(* CODESYS project NPM_v1
   Version: 1.12

Project tree, tasks and I/O mapping:
  _750_8001_WAGO_Basic_Controller_100 : 750-8001 WAGO Basic Controller 100, WAGO, order no. 750-8001, version 1.1.0.1
    application Application
    Kbus : Kbus, WAGO, version 2.1.0.1
        unmapped channels: K-BUS diagnostics
      SC11 : 750-430, WAGO, order no. 750-430, version 2.0.0.14
          unmapped channels: _IN
      SC21 : 750-530, WAGO, order no. 750-530, version 2.0.0.15
          unmapped channels: _OUT
      SC31 : 750-459#08, WAGO, order no. 750-459, version 2.0.0.13
          unmapped channels: _IW 1, _IW 2, _IW 3, _IW 4
      SC32 : 750-459#08, WAGO, order no. 750-459, version 2.0.0.13
          unmapped channels: _IW 1, _IW 2, _IW 3, _IW 4
      SC41 : 750-658#24, WAGO, order no. 750-658, version 2.0.0.11
          unmapped channels: _INPUTCHANNEL, _OUTPUTCHANNEL
      SC42 : 750-658#24, WAGO, order no. 750-658, version 2.0.0.11
          unmapped channels: _INPUTCHANNEL, _OUTPUTCHANNEL
  _750_8212_PFC200 : 750-8212 PFC200, WAGO, order no. 750-8212, version 6.1.1.11
    application Application
      libraries: WagoAppCanLayer2, 1.6.1.4 (WAGO); BASIC, 3.3.4.0 (OSCAT); Util, 3.5.19.0 (System); CAA Memory, * (CAA Technical Workgroup)
      task FastTask (cyclic, interval 1 ms, priority 5) calls CAN_Main
      task Task (cyclic, interval 200 ms, priority 15) calls Simulate, Main
      ALGO/
        SOC/
          global variables gvSOC
          function block SOC [ST]: Calculate, CheckSOCLimits, GetSOCFromCharge, RecalibrateViaLookUpTable
          data type typSOC
        SOF/
          function block CurrentDerating [ST]: Calculate, CalculateCurves, CalculateTemperatureBasedCurrentLimit, CalculateVoltageBasedCurrentLimits, Fb_Init
          global variables gvSOF
          data type typSOF
          data type typSOF_CONFIG
          data type typSOF_CURRENT_LIMITS
          data type typSOF_CURVE
        StateEstimation/
          function block StateEstimation [ST]
      BALANCING/
        function block BAL_Dukosi [ST]: Activate, BalancingAlarm, CheckStateRequest, Deactivate, ProcessState_Balancing, ProcessState_CheckBalancing, Run, SetStateRequest, TransferStateRequest
        global variables BALANCING_CONFIG
        function block BalancingControl [ST]: Activate, CheckStateRequest, Deactivate, Process, ProcessState_Balancing, ProcessState_CheckBalancing, SetStateRequest
        data type eBAL_RETURN
        data type eBAL_STATE
        data type eBAL_STATE_REQUEST
        data type eBAL_SUB_STATE
        global variables gvBALANCING
        data type typBAL_STATE
        data type typBALANCING_CONTROL
      BMS/
        function block StringMinMax [ST]: CalculateDyeTemperatureMinMaxAverage, CalculateTemperatureMinMaxAverage, CalculateVoltageMinMaxAverage, CheckDyeTemperatureSpread, CheckTemperatureSpread, CheckVoltageSpread, Main, ValidateCellDyeTemperature, ValidateCellTemperature, ValidateCellVoltage
      function block BMS_String [ST]: GetCurrentFlowDirection, GetStringState, UpdateStringState
      BMSUtils/
        function DecodeCAN_ID [ST]
        function GetSOCFromVoltage [ST]
      CANBUS/
        function block CAN [ST]: Init, Read, UpdateCellData, Write
        global variables CAN_CONFIG
        program CAN_Main [ST]
        function block CAN_TxCurrentSensor [ST]
        function block CAN_TxDukosi [ST]
        CANUtils/
          function CAN_TO_DINT [ST]
          function CAN_TO_INT [ST]
          function CAN_TO_REAL [ST]
        data type eCAN_MESSAGE_ID
        data type eTX_STATUS
        global variables GVL_CAN_Data
        Queue/
          function block CAN_Queue [ST]: addToQueue, getFront, isEmpty, isFull, removeFromQueue
          interface ICAN_Queue: addToQueue, getFront, isEmpty, isFull, removeFromQueue
        data type typCAN_SIGNAL_RX
        data type typCAN_SIGNAL_RX_CONFIG
        data type typCAN_SIGNAL_RX_INFO
        data type typCAN_SIGNAL_TX
      CONFIG/
        global variables BAT_CELL_CONFIG
        global variables STRING_CONFIG
      data type eCANCommState
      global variables gvBMS
      global variables gvCELLS
      program Main [ST]
      function block Module [ST]
      global variables PersistentVars
      program Simulate [ST]
      data type typCAN_ID
      Types/
        CELL/
          Alarms/
            data type typCELL_ALARM_BITS
            data type uCELL_ALARMS
          Control/
            data type typBAL_CONTROL_BITS
            data type uBAL_CONTROL_BYTE
          Status/
            data type typCELL_BAL_STATUS_BITS
            data type uCELL_BAL_STATUS
          data type typCELL_ALARMS
          data type typCELL_BAL_CURRENT
          data type typCELL_BAL_STATUS
          data type typCELL_CONTROL
          data type typCELL_DYE_TEMPERATURE
          data type typCELL_MEAS
          data type typCELL_MOL_FLAG
          data type typCELL_MSL_FLAG
          data type typCELL_RSL_FLAG
          data type typCELL_TEMP
          data type typCELL_TEMPERATURE
          data type typCELL_VOLTAGE
        data type eBMS_CURRENT_FLOW_STATE
        data type eRET_VAL
        data type eSTRING_STATE
        data type NULL_REF
        data type typERROR_FLAG
        data type typMIN_MAX
        data type typSOE
        data type typSOH
        data type typSTRING_STATE
        data type typSTRING_VALUES
        data type typVoltageVsSOC
      data type typStats
      Utils/
        function BYTE_OF_DWORD [ST]
        function Compare2Arrays [ST]
        function MATH_LinearInterpolation [ST]
        function block Pulse1Sec [ST]
        function Sigmoid [ST]
        function T_PLC_MS [ST]
    Kbus : Kbus, WAGO, version 2.1.0.1
        unmapped channels: K-BUS diagnostics
      _750_658_24 : 750-658#48, WAGO, order no. 750-658, version 2.0.0.11
          unmapped channels: _INPUTCHANNEL, _OUTPUTCHANNEL
      _75x_2DI : 75x-2DI, WAGO, version 2.0.0.13
          unmapped channels: _IN
      _75x_2DO : 75x-2DO, WAGO, version 2.0.0.13
          unmapped channels: _OUT
    Serial
      COM1 : COM1, WAGO, version 0.0.0.19
  text list GlobalTextList
*)

// _750_8212_PFC200/Application/eCANCommState
{attribute 'qualified_only'}
{attribute 'strict'}
TYPE eCANCommState :
(
	INIT,
	OPEN_L2,
	CLOSE_L2,
	RESET_L2,
	CONFIG_L2,
	ALARM,
	READ,
	WRITE
);
END_TYPE

// _750_8212_PFC200/Application/typCAN_ID
TYPE typCAN_ID :
STRUCT
	P : BYTE; //Prority
	//PGN : WORD;
	ID : BYTE; //CAN type
	CA : BYTE; //Cell address
	SA : BYTE; //Station address
END_STRUCT
END_TYPE

// _750_8212_PFC200/Application/typStats
TYPE typStats :
STRUCT
	MinValue : REAL;
	MaxValue : REAL;
	AvgValue : REAL;
END_STRUCT
END_TYPE

// _750_8212_PFC200/Application/BALANCING/eBAL_RETURN
{attribute 'qualified_only'}
{attribute 'strict'}
TYPE eBAL_RETURN :
(
	BAL_OK,               
    BAL_BUSY_OK,           
    BAL_REQUEST_PENDING,   
    BAL_ILLEGAL_REQUEST,   
    BAL_INIT_ERROR, 
    BAL_OK_FROM_ERROR,
    BAL_ERROR,
    BAL_ALREADY_INITIALIZED,
    BAL_ILLEGAL_TASK_TYPE
);
END_TYPE

// _750_8212_PFC200/Application/BALANCING/eBAL_STATE
{attribute 'qualified_only'}
{attribute 'strict'}
TYPE eBAL_STATE :
(
	BAL_STATEMACH_UNINITIALIZED,
    BAL_STATEMACH_INITIALIZATION,
    BAL_STATEMACH_INITIALIZED,
    BAL_STATEMACH_CHECK_BALANCING,
    BAL_STATEMACH_BALANCE,
    BAL_STATEMACH_NO_BALANCING,
    BAL_STATEMACH_ALLOWBALANCING,
    BAL_STATEMACH_GLOBALDISABLE,
    BAL_STATEMACH_GLOBALENABLE,
    BAL_STATEMACH_UNDEFINED,
    BAL_STATEMACH_RESERVED1,
    BAL_STATEMACH_ERROR
);
END_TYPE

// _750_8212_PFC200/Application/BALANCING/eBAL_STATE_REQUEST
{attribute 'qualified_only'}
{attribute 'strict'}
TYPE eBAL_STATE_REQUEST :
(
	BAL_STATE_INIT_REQUEST,     
    BAL_STATE_ERROR_REQUEST,     
    BAL_STATE_NO_BALANCING_REQUEST, 
    BAL_STATE_ALLOWBALANCING_REQUEST, 
    BAL_STATE_GLOBAL_DISABLE_REQUEST,
    BAL_STATE_GLOBAL_ENABLE_REQUEST, 
    BAL_STATE_NO_REQUEST    
);
END_TYPE

// _750_8212_PFC200/Application/BALANCING/eBAL_SUB_STATE
{attribute 'qualified_only'}
{attribute 'strict'}
TYPE eBAL_SUB_STATE :
(
	BAL_ENTRY,       
    BAL_CHECK_IMBALANCES,
    BAL_COMPUTE_IMBALANCES,
    BAL_ACTIVATE_BALANCING,
    BAL_CHECK_LOWEST_VOLTAGE,
    BAL_CHECK_CURRENT
);
END_TYPE

// _750_8212_PFC200/Application/BALANCING/typBAL_STATE
TYPE typBAL_STATE :
STRUCT
	active : BOOL;
	balancingAllowed : BOOL;
	balancingGlobalAllowed : BOOL;
	balancingThreshold : INT;
	state : eBAL_STATE;
	substate : eBAL_SUB_STATE;
	stateRequest : eBAL_STATE_REQUEST;
END_STRUCT
END_TYPE

// _750_8212_PFC200/Application/BALANCING/typBALANCING_CONTROL
TYPE typBALANCING_CONTROL :
STRUCT
	enableBalancing : BOOL;
	threshold_mV : INT;
	request : BOOL;
	balancingState : ARRAY [1..STRING_CONFIG.BS_TOTAL_NR_OF_CELLS] OF INT;
	nrBalancedCells : INT;
END_STRUCT
END_TYPE

// _750_8212_PFC200/Application/CANBUS/eCAN_MESSAGE_ID
{attribute 'qualified_only'}
{attribute 'strict'}
TYPE eCAN_MESSAGE_ID :
(
	NONE,
	CELL_MEAS,
	CELL_TEMP,
	CELL_BAL
)BYTE;
END_TYPE

// _750_8212_PFC200/Application/CANBUS/eTX_STATUS
{attribute 'qualified_only'}
{attribute 'strict'}
TYPE eTX_STATUS :
(
	ST_CAN_TX_INIT, 
  	ST_CAN_TX_NEXT_REQ, 
  	ST_CAN_TX_BUSY, 
  	ST_CAN_TX_WRITE, 
  	ST_TCP_RECV_ERROR
);
END_TYPE

// _750_8212_PFC200/Application/CANBUS/typCAN_SIGNAL_RX
TYPE typCAN_SIGNAL_RX :
STRUCT
	Config : typCAN_SIGNAL_RX_CONFIG;
	Info : typCAN_SIGNAL_RX_INFO;
END_STRUCT
END_TYPE

// _750_8212_PFC200/Application/CANBUS/typCAN_SIGNAL_RX_CONFIG
TYPE typCAN_SIGNAL_RX_CONFIG :
STRUCT
	ID : DWORD;
	Resolution : REAL;
	Offset : REAL;
END_STRUCT
END_TYPE

// _750_8212_PFC200/Application/CANBUS/typCAN_SIGNAL_RX_INFO
TYPE typCAN_SIGNAL_RX_INFO :
STRUCT
	Data : ARRAY [1..8] OF BYTE;
	ReadRX : WagoAppCanLayer2.FbCanRx29BitFrame;
	TimeOutDelay : Standard.TON;
	pktReceived : DINT;
	pktCounter : DINT;
	pktCounter_old : DINT;
	Timpstamp : DWORD;
	previousTimestamp : DWORD;
	deltaT : DWORD;
	read : BOOL;
	newData : BOOL;
	TimeOutAlarm : BOOL;
END_STRUCT
END_TYPE

// _750_8212_PFC200/Application/CANBUS/typCAN_SIGNAL_TX
TYPE typCAN_SIGNAL_TX :
STRUCT
	CAN_NODE : __SYSTEM.IQueryInterface;
	CAN_ID : WORD;
	Data : ARRAY [1..8] OF BYTE;
END_STRUCT
END_TYPE

// _750_8212_PFC200/Application/Types/eBMS_CURRENT_FLOW_STATE
{attribute 'qualified_only'}
{attribute 'strict'}
TYPE eBMS_CURRENT_FLOW_STATE :
(
	AT_REST,
	RELAXATION,
	CHARGING,
	DISCHARGING
);
END_TYPE

// _750_8212_PFC200/Application/Types/eRET_VAL
{attribute 'qualified_only'}
{attribute 'strict'}
TYPE eRET_VAL :
(
	STD_OK,
	STD_NOT_OK
);
END_TYPE

// _750_8212_PFC200/Application/Types/eSTRING_STATE
{attribute 'qualified_only'}
{attribute 'strict'}
TYPE eSTRING_STATE :
(
	CHARGING,
	DISCHARGING,
	RELAXATION,
	AT_REST
);
END_TYPE

// _750_8212_PFC200/Application/Types/NULL_REF
TYPE NULL_REF : LINT :=0; END_TYPE

// _750_8212_PFC200/Application/Types/typERROR_FLAG
TYPE typERROR_FLAG :
STRUCT
END_STRUCT
END_TYPE

// _750_8212_PFC200/Application/Types/typMIN_MAX
TYPE typMIN_MAX :
STRUCT
	averageCellVoltage_mV : REAL;
	minimumCellVoltage_mV : REAL;
	maximumCellVoltage_mV : REAL;
	averageTemperature_degC : REAL;
	minimumTemperature_degC : REAL;
	maximumTemperature_degC : REAL;
	averageDyeTemperature_degC : REAL;
	minimumDyeTemperature_degC : REAL;
	maximumDyeTemperature_degC : REAL;
	validMeasuredCellTemperatures : INT;
	validMeasuredCellDyeTemperatures : INT;
	validMeasuredCellVoltages : INT;

END_STRUCT
END_TYPE

// _750_8212_PFC200/Application/Types/typSOE
TYPE typSOE :
STRUCT
	averageSOE_pct : REAL;
	minimumSOE_pct : REAL;
	maximumSOE_pct : REAL;
	averageSOE_Wh : REAL;
	minimumSOE_Wh : REAL;
	maximumSOE_Wh : REAL;
END_STRUCT
END_TYPE

// _750_8212_PFC200/Application/Types/typSOH
TYPE typSOH :
STRUCT
	averageSOH_pct : REAL;
	minimumSOH_pct : REAL;
	maximumSOH_pct : REAL;
END_STRUCT
END_TYPE

// _750_8212_PFC200/Application/Types/typSTRING_STATE
TYPE typSTRING_STATE :
STRUCT
	currentFlowState : eBMS_CURRENT_FLOW_STATE;
	restTime : INT;
END_STRUCT
END_TYPE

// _750_8212_PFC200/Application/Types/typSTRING_VALUES
TYPE typSTRING_VALUES :
STRUCT
	StringCurrent : REAL;
	StringVoltage : REAL;
	StringTemperature : REAL;
	StringPower : REAL;
END_STRUCT
END_TYPE

// _750_8212_PFC200/Application/Types/typVoltageVsSOC
TYPE typVoltageVsSOC :
STRUCT
	Voltage : INT;
	SOC : REAL;
END_STRUCT
END_TYPE

// _750_8212_PFC200/Application/ALGO/SOC/typSOC
TYPE typSOC :
STRUCT
	averageSOC_pct : REAL;
	minimumSOC_pct : REAL;
	maximumSOC_pct : REAL;
END_STRUCT
END_TYPE

// _750_8212_PFC200/Application/ALGO/SOF/typSOF
TYPE typSOF :
STRUCT
	recommandedContinuosChargeCurrent : REAL;
	recommandedContinuosDischargeCurrent : REAL;
	recommandedPeakChargeCurrent : REAL;
	recommandedPeakDischargeCurrent : REAL;
END_STRUCT
END_TYPE

// _750_8212_PFC200/Application/ALGO/SOF/typSOF_CONFIG
TYPE typSOF_CONFIG :
STRUCT
    maximumDischargeCurrent_mA : REAL;
    maximumChargeCurrent_mA : REAL;
    limpCurrent_mA : REAL;

    cutoffLowTemperatureDischarge_degC : REAL;
    limitLowTemperatureDischarge_degC : REAL;
    cutoffLowTemperatureCharge_degC : REAL;
    limitLowTemperatureCharge_degC : REAL;
    

    cutoffHighTemperatureDischarge_degC : REAL;
    limitHighTemperatureDischarge_degC : REAL;
    cutoffHighTemperatureCharge_degC : REAL;
    limitHighTemperatureCharge_degC : REAL;
    

    cutoffUpperCellVoltage_mV : REAL;
    limitUpperCellVoltage_mV : REAL;
    cutoffLowerCellVoltage_mV : REAL;
    limitLowerCellVoltage_mV : REAL;
END_STRUCT
END_TYPE

// _750_8212_PFC200/Application/ALGO/SOF/typSOF_CURRENT_LIMITS
TYPE typSOF_CURRENT_LIMITS :
STRUCT
	ContinuosChargeCurrent : REAL;
	ContinuosDischargeCurrent : REAL;
	PeakChargeCurrent : REAL;
	PeakDischargeCurrent : REAL;
END_STRUCT
END_TYPE

// _750_8212_PFC200/Application/ALGO/SOF/typSOF_CURVE
TYPE typSOF_CURVE :
STRUCT
	slopeLowTemperatureDischarge : REAL;   
    offsetLowTemperatureDischarge : REAL;  
    slopeHighTemperatureDischarge : REAL;  
    offsetHighTemperatureDischarge : REAL; 
    
    slopeLowTemperatureCharge : REAL;   
    offsetLowTemperatureCharge : REAL;  
    slopeHighTemperatureCharge : REAL;  
    offsetHighTemperatureCharge : REAL; 
    
    slopeUpperCellVoltage : REAL;  
    offsetUpperCellVoltage : REAL; 
    slopeLowerCellVoltage : REAL;  
    offsetLowerCellVoltage : REAL; 
END_STRUCT
END_TYPE

// _750_8212_PFC200/Application/Types/CELL/typCELL_ALARMS
TYPE typCELL_ALARMS :
STRUCT
	cellStatus : ARRAY [1..STRING_CONFIG.BS_TOTAL_NR_OF_CELLS] OF uCELL_ALARMS;
	//timeStamp : ARRAY [1..STRING_CONFIG.BS_NR_OF_MODULES, 1..STRING_CONFIG.BS_TOTAL_NR_OF_CELLS] OF DINT;
	//previousTimeStamp : ARRAY [1..STRING_CONFIG.BS_NR_OF_MODULES, 1..STRING_CONFIG.BS_TOTAL_NR_OF_CELLS] OF DINT;
END_STRUCT
END_TYPE

// _750_8212_PFC200/Application/Types/CELL/typCELL_BAL_CURRENT
TYPE typCELL_BAL_CURRENT :
STRUCT
	cellBalCurrent_mAmps : ARRAY [1..STRING_CONFIG.BS_TOTAL_NR_OF_CELLS] OF INT;
	//invalidCellBalCurrent : ARRAY [1..STRING_CONFIG.BS_NR_OF_MODULES] OF BOOL;
	nrValidCellBalCurrent : INT;
	//timeStamp : ARRAY [1..STRING_CONFIG.BS_NR_OF_MODULES, 1..STRING_CONFIG.BS_TOTAL_NR_OF_CELLS] OF DINT;
	//previousTimeStamp : ARRAY [1..STRING_CONFIG.BS_NR_OF_MODULES, 1..STRING_CONFIG.BS_TOTAL_NR_OF_CELLS] OF DINT;
END_STRUCT
END_TYPE

// _750_8212_PFC200/Application/Types/CELL/typCELL_BAL_STATUS
TYPE typCELL_BAL_STATUS :
STRUCT
	cellBalStatus : ARRAY [1..STRING_CONFIG.BS_TOTAL_NR_OF_CELLS] OF uCELL_BAL_STATUS;
	//timeStamp : ARRAY [1..STRING_CONFIG.BS_NR_OF_MODULES, 1..STRING_CONFIG.BS_TOTAL_NR_OF_CELLS] OF DINT;
	//previousTimeStamp : ARRAY [1..STRING_CONFIG.BS_NR_OF_MODULES, 1..STRING_CONFIG.BS_TOTAL_NR_OF_CELLS] OF DINT;
END_STRUCT
END_TYPE

// _750_8212_PFC200/Application/Types/CELL/typCELL_CONTROL
TYPE typCELL_CONTROL :
STRUCT
	BAL_tgtVoltage : ARRAY [1..STRING_CONFIG.BS_TOTAL_NR_OF_CELLS] OF INT;
	BAL_loadResistor : ARRAY [1..STRING_CONFIG.BS_TOTAL_NR_OF_CELLS] OF INT;
	BAL_dutyCycle : ARRAY [1..STRING_CONFIG.BS_TOTAL_NR_OF_CELLS] OF BYTE;
	BAL_watchdogUnit : ARRAY [1..STRING_CONFIG.BS_TOTAL_NR_OF_CELLS] OF BYTE;
	BAL_watchdogCounter : ARRAY [1..STRING_CONFIG.BS_TOTAL_NR_OF_CELLS] OF BYTE;
	BAL_Control : ARRAY [1..STRING_CONFIG.BS_TOTAL_NR_OF_CELLS] OF uBAL_CONTROL_BYTE;
	timeStamp : ARRAY [1..STRING_CONFIG.BS_TOTAL_NR_OF_CELLS] OF DINT;
	previousTimeStamp : ARRAY [1..STRING_CONFIG.BS_TOTAL_NR_OF_CELLS] OF DINT;
END_STRUCT
END_TYPE

// _750_8212_PFC200/Application/Types/CELL/typCELL_DYE_TEMPERATURE
TYPE typCELL_DYE_TEMPERATURE :
STRUCT
	cellDyeTemperature_deg : ARRAY [1..STRING_CONFIG.BS_TOTAL_NR_OF_CELLS] OF INT;
	invalidCellDyeTemperature : ARRAY [1..STRING_CONFIG.BS_NR_OF_MODULES] OF ULINT;
	nrValidCellDyeTemperatures :  INT;
	//timeStamp : ARRAY [1..STRING_CONFIG.BS_NR_OF_MODULES, 1..STRING_CONFIG.BS_TOTAL_NR_OF_CELLS] OF DINT;
	//previousTimeStamp : ARRAY [1..STRING_CONFIG.BS_NR_OF_MODULES, 1..STRING_CONFIG.BS_TOTAL_NR_OF_CELLS] OF DINT;
END_STRUCT
END_TYPE

// _750_8212_PFC200/Application/Types/CELL/typCELL_MEAS
TYPE typCELL_MEAS :
STRUCT
	voltage : typCELL_VOLTAGE;
	balCurrent : typCELL_BAL_CURRENT;
	cellStatus : ARRAY [1..STRING_CONFIG.BS_TOTAL_NR_OF_CELLS] OF uCELL_ALARMS;
	cellBalStatus : ARRAY [1..STRING_CONFIG.BS_TOTAL_NR_OF_CELLS] OF uCELL_BAL_STATUS;
	timeStamp : ARRAY [1..STRING_CONFIG.BS_TOTAL_NR_OF_CELLS] OF DWORD;
	previousTimeStamp : ARRAY [1..STRING_CONFIG.BS_TOTAL_NR_OF_CELLS] OF DWORD;
END_STRUCT
END_TYPE

// _750_8212_PFC200/Application/Types/CELL/typCELL_MOL_FLAG
(*Maximum operating limis*)
TYPE typCELL_MOL_FLAG :
STRUCT
	overVoltage 				: BOOL;
	underVoltage 				: BOOL;
	overTemperatureCharge 		: BOOL;
	overTemperatureDischarge 	: BOOL;
	underTemperatureCharge 		: BOOL;
	underTemperatureDischarge 	: BOOL;
	ChargeOvercurrent 			: BOOL;
	DischargeOvercurrent 		: BOOL;
END_STRUCT
END_TYPE

// _750_8212_PFC200/Application/Types/CELL/typCELL_MSL_FLAG
(*Maximum saftey limits*)
TYPE typCELL_MSL_FLAG :
STRUCT
	overVoltage 				: BOOL;
	underVoltage 				: BOOL;
	overTemperatureCharge 		: BOOL;
	overTemperatureDischarge 	: BOOL;
	underTemperatureCharge 		: BOOL;
	underTemperatureDischarge 	: BOOL;
	ChargeOvercurrent 			: BOOL;
	DischargeOvercurrent 		: BOOL;
END_STRUCT
END_TYPE

// _750_8212_PFC200/Application/Types/CELL/typCELL_RSL_FLAG
(*Recomanded saftey limits*)
TYPE typCELL_RSL_FLAG :
STRUCT
	overVoltage 				: BOOL;
	underVoltage 				: BOOL;
	overTemperatureCharge 		: BOOL;
	overTemperatureDischarge 	: BOOL;
	underTemperatureCharge 		: BOOL;
	underTemperatureDischarge 	: BOOL;
	ChargeOvercurrent 			: BOOL;
	DischargeOvercurrent 		: BOOL;
END_STRUCT
END_TYPE

// _750_8212_PFC200/Application/Types/CELL/typCELL_TEMP
TYPE typCELL_TEMP :
STRUCT
	temperature : typCELL_TEMPERATURE;
	dyeTemperature : typCELL_DYE_TEMPERATURE;
	timeStamp : ARRAY [1..STRING_CONFIG.BS_TOTAL_NR_OF_CELLS] OF DWORD;
	previousTimeStamp : ARRAY [1..STRING_CONFIG.BS_TOTAL_NR_OF_CELLS] OF DWORD;
END_STRUCT
END_TYPE

// _750_8212_PFC200/Application/Types/CELL/typCELL_TEMPERATURE
TYPE typCELL_TEMPERATURE :
STRUCT
	cellTemperature_deg : ARRAY [1..STRING_CONFIG.BS_TOTAL_NR_OF_CELLS] OF INT;
	invalidCellTemperature : ARRAY [1..STRING_CONFIG.BS_NR_OF_MODULES] OF ULINT;
	nrValidCellTemperatures :  INT;
	//timeStamp : ARRAY [1..STRING_CONFIG.BS_NR_OF_MODULES, 1..STRING_CONFIG.BS_TOTAL_NR_OF_CELLS] OF DINT;
	//previousTimeStamp : ARRAY [1..STRING_CONFIG.BS_NR_OF_MODULES, 1..STRING_CONFIG.BS_TOTAL_NR_OF_CELLS] OF DINT;
END_STRUCT
END_TYPE

// _750_8212_PFC200/Application/Types/CELL/typCELL_VOLTAGE
TYPE typCELL_VOLTAGE :
STRUCT
	stringVoltage_mV : DINT;
	//moduleVoltage_mV : ARRAY [1..STRING_CONFIG.BS_NR_OF_MODULES] OF DINT;
	cellVoltage_mV : ARRAY [1..STRING_CONFIG.BS_TOTAL_NR_OF_CELLS] OF INT;
	invalidCellVoltage : ARRAY [1..STRING_CONFIG.BS_NR_OF_MODULES] OF ULINT;
	nrValidCellVoltages : INT;
	//timeStamp : ARRAY [1..STRING_CONFIG.BS_NR_OF_MODULES, 1..STRING_CONFIG.BS_TOTAL_NR_OF_CELLS] OF DINT;
	//previousTimeStamp : ARRAY [1..STRING_CONFIG.BS_NR_OF_MODULES, 1..STRING_CONFIG.BS_TOTAL_NR_OF_CELLS] OF DINT;
END_STRUCT
END_TYPE

// _750_8212_PFC200/Application/Types/CELL/Alarms/typCELL_ALARM_BITS
TYPE typCELL_ALARM_BITS :
STRUCT
	LIM_V_MAX_OP : BIT; //Maximum operating voltage limit
	LIM_V_MIN_OP : BIT; //Minimum operating voltage limit
	LIM_V_MAX_SAFETY : BIT; //Maximum safety voltage limit
	LIM_V_MIN_SAFETY : BIT; //Minimum safety voltage limi
// 	LIM_I_DISCHARGE_DC : BIT; //Discharge current DC limit
// 	LIM_I_CHARGE_DC : BIT; //Charge current DC limit
// 	LIM_I_DISCHARGE_PULSE : BIT; //Discharge current pulse limit
// 	LIM_I_CHARGE_PULSE : BIT; //Charge current pulse limit
// 	LIM_I_DISCHARGE_PEAK : BIT; //Discharge current peak limit
// 	LIM_I_CHARGE_PEAK : BIT; //Charge current peak limit
// 	LIM_MEASUREMENT_PWM_IN_CURRENT : BIT; //Limit for measurement type PWM_IN_CURRENT
	LIM_MEASUREMENT_THERM1 : BIT; //Limit for measurement type THERM1
	HVIL_CONTACT: BIT; //HVIL_Contact
	LIM_MEASUREMENT_DTS : BIT; //Limit for measurement type DTS
	LIM_MEASUREMENT_PWM_IN_VOLTAGE : BIT; //Limit for measurement type PWM_IN_VOLTAGE
	LIM_OTHERS : BIT; //Other alarms
END_STRUCT
END_TYPE

// _750_8212_PFC200/Application/Types/CELL/Alarms/uCELL_ALARMS
TYPE uCELL_ALARMS :
UNION
	AlarmWord : WORD;
	CellAlarms : typCELL_ALARM_BITS;
END_UNION
END_TYPE

// _750_8212_PFC200/Application/Types/CELL/Control/typBAL_CONTROL_BITS
TYPE typBAL_CONTROL_BITS :
STRUCT
	BAL_enTgtVoltage : BIT; //Enable target voltage
	BAL_externalFET  : BIT; //Use external FET
END_STRUCT
END_TYPE

// _750_8212_PFC200/Application/Types/CELL/Control/uBAL_CONTROL_BYTE
TYPE uBAL_CONTROL_BYTE :
UNION
	ControlByte : BYTE;
	ControlBits : typBAL_CONTROL_BITS;
END_UNION
END_TYPE

// _750_8212_PFC200/Application/Types/CELL/Status/typCELL_BAL_STATUS_BITS
TYPE typCELL_BAL_STATUS_BITS :
STRUCT
	BAL_isActive 		: BIT; //Cell balancing in active state 
	BAL_IsStopCmd 		: BIT; //Cell balancing stopped due to balance stop command
	BAL_IsStopTgtVolt 	: BIT; //Cell balancing stopped due to target voltage reached
	BAL_isStopTgtSoc 	: BIT; //Cell balancing stopped due to target SoC reached
	BAL_isStopTgtWh 	: BIT; //Cell balancing stopped due to target watt hours reached
	BAL_isStopError 	: BIT; //Cell balancing stopped due to an error
	BAL_isStopTemp 		: BIT; //Cell balancing stopped due to an over temperature error
	BAL_isStopOther 	: BIT; //Cell balancing stopped due to any other error
END_STRUCT
END_TYPE

// _750_8212_PFC200/Application/Types/CELL/Status/uCELL_BAL_STATUS
TYPE uCELL_BAL_STATUS :
STRUCT
	StatusWord : WORD;
	BalStatus : typCELL_BAL_STATUS_BITS;
END_STRUCT
END_TYPE

// _750_8212_PFC200/Application/gvBMS
{attribute 'qualified_only'}
VAR_GLOBAL
	gvMinMax : typMIN_MAX;
	gcStringValues : typSTRING_VALUES;
	gcStringState : typSTRING_STATE;
	Fb_String : BMS_String := (StringState := gcStringState);
	StringStat : StringMinMax := (MinMaxTable := gvMinMax);
	BalancingControl : BAL_Dukosi := (DKS_BALControl := gvCells.gvCellControl, DKS_BALCurrent := gvCells.gvCellMeas.balCurrent, DKS_BALStatus := gvCells.gvCellMeas,
									  DKS_CellVoltage := gvCells.gvCellMeas.voltage, DKS_MinMax := gvMinMax, balControl := gvBalancing.gvBALANCING_CONTROL);
	
	
	Pulse1Sec : Pulse1Sec;
	
	
	
END_VAR

// _750_8212_PFC200/Application/gvCELLS
{attribute 'qualified_only'}
VAR_GLOBAL
	//Cells : typCELLS_VALUES;
	gvCellMeas : typCELL_MEAS;
	gvCellTemp : typCELL_TEMP;
	gvCellControl : typCELL_CONTROL;
// 	gvCellVoltages : typCELL_VOLTAGE;
// 	gvCellTemperatures : typCELL_TEMPERATURE;
// 	gvCellDyeTemperatures : typCELL_DYE_TEMPERATURE;
// 	gvCellAlarms : typCELL_ALARMS_1;
END_VAR

// _750_8212_PFC200/Application/PersistentVars
{attribute 'qualified_only'}
VAR_GLOBAL PERSISTENT RETAIN
	SOC : typSOC;
END_VAR

// _750_8212_PFC200/Application/BALANCING/BALANCING_CONFIG
{attribute 'qualified_only'}
VAR_GLOBAL CONSTANT
	//default value for the BAL voltage threshold 
	BAL_DEFAULT_THRESHOLD_mV : INT := 200;

	//maximum value that BAL voltage threshold may take
	BAL_MAXIMUM_THRESHOLD_mV : INT := 5000;
	
	//minimum value that BAL voltage threshold may take
	BAL_MINIMUM_THRESHOLD_mV : INT := 0; 
	
	//BAL hysteresis for voltage threshold when balancing was finished in mV
	BAL_HYSTERESIS_mV : INT := 200;
	
	//BAL lower voltage limit in MV
	BAL_LOWER_VOLTAGE_LIMIT_mV : INT := 2000;
	
	//BAL upper temperature limit
	BAL_UPPER_TEMPERATURE_LIMIT_degC : INT := 70;
	
END_VAR

// _750_8212_PFC200/Application/BALANCING/gvBALANCING
{attribute 'qualified_only'}
VAR_GLOBAL
	gvBALANCING_CONTROL : typBALANCING_CONTROL;
END_VAR

// _750_8212_PFC200/Application/CANBUS/CAN_CONFIG
{attribute 'qualified_only'}
{attribute 'global_init_slot' := '49988'}
VAR_GLOBAL
	CAN_OFFSET : DWORD := 16#80000000;
	CAN_TIMEOUT_DELAY : TIME := T#2S;
END_VAR

// _750_8212_PFC200/Application/CANBUS/GVL_CAN_Data
VAR_GLOBAL

	// typCanLayer2RxAllSchedule : typCanLayer2RxSchedule;
	arrCANDataRX: ARRAY [1..STRING_CONFIG.BS_TOTAL_NR_OF_CELLS] OF typCAN_SIGNAL_RX := [(Config := (ID := 16#98FF0101)),
																						 (Config := (ID := 16#98FF0301)),
																						 (Config := (ID := 16#98FF0501)),
																						 (Config := (ID := 16#98FF0701)),
																						 (Config := (ID := 16#98FF0901)),
																						 (Config := (ID := 16#98FF0B01)),
																						 (Config := (ID := 16#98FF0D01)),
																						 (Config := (ID := 16#98FF0F01)),
																						 (Config := (ID := 16#98FF1101)),
																						 (Config := (ID := 16#98FF1301)),
																						 (Config := (ID := 16#98FF1501)),
																						 (Config := (ID := 16#98FF1701)),
																						 (Config := (ID := 16#98FF1901)),
																						 (Config := (ID := 16#98FF1B01)),
																						 (Config := (ID := 16#98FF1D01)),
																						 (Config := (ID := 16#98FF1F01)),
																						 (Config := (ID := 16#98FF2101)),
																						 (Config := (ID := 16#98FF2301)),
																						 (Config := (ID := 16#98FF2501)),
																						 (Config := (ID := 16#98FF2701)),
																						 (Config := (ID := 16#98FF2901)),
																						 (Config := (ID := 16#98FF2B01)),
																						 (Config := (ID := 16#98FF2D01)),
																						 (Config := (ID := 16#98FF2F01)),
																						 (Config := (ID := 16#98FF3101)),
																						 (Config := (ID := 16#98FF3301)),
																						 (Config := (ID := 16#98FF3501)),
																						 (Config := (ID := 16#98FF3701)),
																						 (Config := (ID := 16#98FF3901)),
																						 (Config := (ID := 16#98FF3B01)),
																						 (Config := (ID := 16#98FF3D01)),
																						 (Config := (ID := 16#98FF3F01)),
																						 (Config := (ID := 16#98FF4101)),
																						 (Config := (ID := 16#98FF4301)),
																						 (Config := (ID := 16#98FF4501)),
																						 (Config := (ID := 16#98FF4701)),
																						 (Config := (ID := 16#98FF4901)),
																						 (Config := (ID := 16#98FF4B01)),
																						 (Config := (ID := 16#98FF4D01)),
																						 (Config := (ID := 16#98FF4F01)),
																						 (Config := (ID := 16#98FF5101)),
																						 (Config := (ID := 16#98FF5301)),
																						 (Config := (ID := 16#98FF5501)),
																						 (Config := (ID := 16#98FF5701)),
																						 (Config := (ID := 16#98FF5901)),
																						 (Config := (ID := 16#98FF5B01)),
																						 (Config := (ID := 16#98FF5D01)),
																						 (Config := (ID := 16#98FF5F01)),
																						 (Config := (ID := 16#98FF6101)),
																						 (Config := (ID := 16#98FF6301)),
																						 (Config := (ID := 16#98FF6501)),
																						 (Config := (ID := 16#98FF6701)),
																						 (Config := (ID := 16#98FF6901)),
																						 (Config := (ID := 16#98FF6B01)),
																						 (Config := (ID := 16#98FF6D01)),
																						 (Config := (ID := 16#98FF6F01)),
																						 (Config := (ID := 16#98FF7101)),
																						 (Config := (ID := 16#98FF7301)),
																						 (Config := (ID := 16#98FF7501)),
																						 (Config := (ID := 16#98FF7701)),
																						 (Config := (ID := 16#98FF7901)),
																						 (Config := (ID := 16#98FF7B01)),
																						 (Config := (ID := 16#98FF7D01)),
																						 (Config := (ID := 16#98FF7F01)),
																						 (Config := (ID := 16#98FF0301)),
																						 (Config := (ID := 16#98FF0501)),
																						 (Config := (ID := 16#98FF0701)),
																						 (Config := (ID := 16#98FF0901)),
																						 (Config := (ID := 16#98FF0B01)),
																						 (Config := (ID := 16#98FF0D01)),
																						 (Config := (ID := 16#98FF0F01)),
																						 (Config := (ID := 16#98FF1101)),
																						 (Config := (ID := 16#98FF1301)),
																						 (Config := (ID := 16#98FF1501)),
																						 (Config := (ID := 16#98FF1701)),
																						 (Config := (ID := 16#98FF1901)),
																						 (Config := (ID := 16#98FF1B01)),
																						 (Config := (ID := 16#98FF1D01)),
																						 (Config := (ID := 16#98FF1F01)),
																						 (Config := (ID := 16#98FF2101)),
																						 (Config := (ID := 16#98FF2301)),
																						 (Config := (ID := 16#98FF2501)),
																						 (Config := (ID := 16#98FF2701)),
																						 (Config := (ID := 16#98FF2901)),
																						 (Config := (ID := 16#98FF2B01)),
																						 (Config := (ID := 16#98FF2D01)),
																						 (Config := (ID := 16#98FF2F01)),
																						 (Config := (ID := 16#98FF3101)),
																						 (Config := (ID := 16#98FF3301)),
																						 (Config := (ID := 16#98FF3501)),
																						 (Config := (ID := 16#98FF3701)),
																						 (Config := (ID := 16#98FF3901)),
																						 (Config := (ID := 16#98FF3B01)),
																						 (Config := (ID := 16#98FF3D01)),
																						 (Config := (ID := 16#98FF3F01)),
																						 (Config := (ID := 16#98FF4101)),
																						 (Config := (ID := 16#98FF4301)),
																						 (Config := (ID := 16#98FF4501)),
																						 (Config := (ID := 16#98FF4701)),
																						 (Config := (ID := 16#98FF4901)),
																						 (Config := (ID := 16#98FF4B01)),
																						 (Config := (ID := 16#98FF4D01)),
																						 (Config := (ID := 16#98FF4F01)),
																						 (Config := (ID := 16#98FF5101)),
																						 (Config := (ID := 16#98FF5301)),
																						 (Config := (ID := 16#98FF5501)),
																						 (Config := (ID := 16#98FF5701)),
																						 (Config := (ID := 16#98FF5901)),
																						 (Config := (ID := 16#98FF5B01)),
																						 (Config := (ID := 16#98FF5D01)),
																						 (Config := (ID := 16#98FF5F01)),
																						 (Config := (ID := 16#98FF6101)),
																						 (Config := (ID := 16#98FF6301)),
																						 (Config := (ID := 16#98FF6501)),
																						 (Config := (ID := 16#98FF6701)),
																						 (Config := (ID := 16#98FF6901)),
																						 (Config := (ID := 16#98FF6B01)),
																						 (Config := (ID := 16#98FF6D01)),
																						 (Config := (ID := 16#98FF6F01)),
																						 (Config := (ID := 16#98FF7101)),
																						 (Config := (ID := 16#98FF7301)),
																						 (Config := (ID := 16#98FF7501)),
																						 (Config := (ID := 16#98FF7701)),
																						 (Config := (ID := 16#98FF7901)),
																						 (Config := (ID := 16#98FF7B01)),
																						 (Config := (ID := 16#98FF7D01)),
																						 (Config := (ID := 16#98FF7F01)),
																						 (Config := (ID := 16#98FF0301)),
																						 (Config := (ID := 16#98FF0501)),
																						 (Config := (ID := 16#98FF0701)),
																						 (Config := (ID := 16#98FF0901)),
																						 (Config := (ID := 16#98FF0B01)),
																						 (Config := (ID := 16#98FF0D01)),
																						 (Config := (ID := 16#98FF0F01)),
																						 (Config := (ID := 16#98FF1101)),
																						 (Config := (ID := 16#98FF1301)),
																						 (Config := (ID := 16#98FF1501)),
																						 (Config := (ID := 16#98FF1701)),
																						 (Config := (ID := 16#98FF1901)),
																						 (Config := (ID := 16#98FF1B01)),
																						 (Config := (ID := 16#98FF1D01)),
																						 (Config := (ID := 16#98FF1F01)),
																						 (Config := (ID := 16#98FF2101)),
																						 (Config := (ID := 16#98FF2301)),
																						 (Config := (ID := 16#98FF2501)),
																						 (Config := (ID := 16#98FF2701)),
																						 (Config := (ID := 16#98FF2901)),
																						 (Config := (ID := 16#98FF2B01)),
																						 (Config := (ID := 16#98FF2D01)),
																						 (Config := (ID := 16#98FF2F01)),
																						 (Config := (ID := 16#98FF3101)),
																						 (Config := (ID := 16#98FF3301)),
																						 (Config := (ID := 16#98FF3501)),
																						 (Config := (ID := 16#98FF3701)),
																						 (Config := (ID := 16#98FF3901)),
																						 (Config := (ID := 16#98FF3B01)),
																						 (Config := (ID := 16#98FF3D01)),
																						 (Config := (ID := 16#98FF3F01)),
																						 (Config := (ID := 16#98FF4101)),
																						 (Config := (ID := 16#98FF4301)),
																						 (Config := (ID := 16#98FF4501)),
																						 (Config := (ID := 16#98FF4701)),
																						 (Config := (ID := 16#98FF4901)),
																						 (Config := (ID := 16#98FF4B01)),
																						 (Config := (ID := 16#98FF4D01)),
																						 (Config := (ID := 16#98FF4F01)),
																						 (Config := (ID := 16#98FF5101)),
																						 (Config := (ID := 16#98FF5301)),
																						 (Config := (ID := 16#98FF5501)),
																						 (Config := (ID := 16#98FF5701)),
																						 (Config := (ID := 16#98FF5901)),
																						 (Config := (ID := 16#98FF5B01)),
																						 (Config := (ID := 16#98FF5D01)),
																						 (Config := (ID := 16#98FF5F01)),
																						 (Config := (ID := 16#98FF6101)),
																						 (Config := (ID := 16#98FF6301)),
																						 (Config := (ID := 16#98FF6501)),
																						 (Config := (ID := 16#98FF6701)),
																						 (Config := (ID := 16#98FF6901)),
																						 (Config := (ID := 16#98FF6B01)),
																						 (Config := (ID := 16#98FF6D01)),
																						 (Config := (ID := 16#98FF6F01)),
																						 (Config := (ID := 16#98FF7101)),
																						 (Config := (ID := 16#98FF7301)),
																						 (Config := (ID := 16#98FF7501)),
																						 (Config := (ID := 16#98FF7701)),
																						 (Config := (ID := 16#98FF7901)),
																						 (Config := (ID := 16#98FF7B01)),
																						 (Config := (ID := 16#98FF7D01)),
																						 (Config := (ID := 16#98FF7F01)),
																						 (Config := (ID := 16#98FF0301)),
																						 (Config := (ID := 16#98FF0501)),
																						 (Config := (ID := 16#98FF0701)),
																						 (Config := (ID := 16#98FF0901)),
																						 (Config := (ID := 16#98FF0B01)),
																						 (Config := (ID := 16#98FF0D01)),
																						 (Config := (ID := 16#98FF0F01)),
																						 (Config := (ID := 16#98FF1101)),
																						 (Config := (ID := 16#98FF1301)),
																						 (Config := (ID := 16#98FF1501)),
																						 (Config := (ID := 16#98FF1701)),
																						 (Config := (ID := 16#98FF1901)),
																						 (Config := (ID := 16#98FF1B01)),
																						 (Config := (ID := 16#98FF1D01))];								
	
END_VAR

// _750_8212_PFC200/Application/CONFIG/BAT_CELL_CONFIG
{attribute 'qualified_only'}
VAR_GLOBAL CONSTANT
	stateOfChargeLookupTable : ARRAY [1..10] OF typVoltageVsSOC;
	stateOfChargeLookupTableSize : UINT := SIZEOF(stateOfChargeLookupTable)/ SIZEOF(typVoltageVsSOC);
	
	CELL_TEMPERATURE_SPREAD_TOLERANCE : REAL := 10;
	CELL_VOLTAGE_SPREAD_TOLERANCE : REAL := 10;
	CELL_DYE_TEMPERATURE_SPREAD_TOLERANCE : REAL := 10;
	
	CURRENT_LEAK : REAL := 1E-6;
	CELL_NOMINAL_CAPACITY_Ah : REAL := 175; //Amps/h
	CELL_NOMINAL_ENERGY_Wh : REAL := 175; //Amps/h
	CELL_NOMINAL_CAPACITY_W : REAL := 955; //W
	CELL_NOMINAL_VOLTAGE_mV : REAL := 2300; //mW
	
	
	(*When maximum safety limit (MSL) is violated, error state is
    requested and contactors will open. When recommended safety limit
    (RSL) or maximum operating limit (MOL) is violated, the respective
    flag will be set.*)
	
	//Maximum temperature limit during discharge.
	CELL_TEMPERATURE_MAX_DISCHARGE_MSL_degC : REAL := 40;
	CELL_TEMPERATURE_MAX_DISCHARGE_RSL_degC : REAL := 39;
	CELL_TEMPERATURE_MAX_DISCHARGE_MOL_degC : REAL := 38;
	
	//Minimum temperature limit during discharge.
	CELL_TEMPERATURE_MIN_DISCHARGE_MSL_degC : REAL := -20;
	CELL_TEMPERATURE_MIN_DISCHARGE_RSL_degC : REAL := -15;
	CELL_TEMPERATURE_MIN_DISCHARGE_MOL_degC : REAL := -10;
	
	//Maximum temperature limit during charge.
	CELL_TEMPERATURE_MAX_CHARGE_MSL_degC : REAL := 40;
	CELL_TEMPERATURE_MAX_CHARGE_RSL_degC : REAL := 39;
	CELL_TEMPERATURE_MAX_CHARGE_MOL_degC : REAL := 38;
	
	//Minimum temperature limit during charge.
	CELL_TEMPERATURE_MIN_CHARGE_MSL_degC : REAL := -20;
	CELL_TEMPERATURE_MIN_CHARGE_RSL_degC : REAL := -15;
	CELL_TEMPERATURE_MIN_CHARGE_MOL_degC : REAL := -10;
	
	//Maximum voltage limit
	CELL_VOLTAGE_MAX_MSL_mV : REAL := 2750;
	CELL_VOLTAGE_MAX_RSL_mV : REAL := 2730;
	CELL_VOLTAGE_MAX_MOL_mV : REAL := 2700;
	
	//Minimum voltage limit
	CELL_VOLTAGE_MIN_MSL_mV : REAL := 2750;
	CELL_VOLTAGE_MIN_RSL_mV : REAL := 2730;
	CELL_VOLTAGE_MIN_MOL_mV : REAL := 2700;
	
	//Deep-discharge cell voltage limit.
	CELL_VOLTAGE_DEEP_DISCHARGE_mV : REAL := CELL_VOLTAGE_MIN_MSL_mV;
	
	//Maximum discharge current limit.
	CELL_CURRENT_MAX_DISCHARGE_MSL_mA : REAL := 175000;
	CELL_CURRENT_MAX_DISCHARGE_RSL_mA : REAL := 175000;
	CELL_CURRENT_MAX_DISCHARGE_MOL_mA : REAL := 175000;
	
	//Maximum charge current limit.
	CELL_CURRENT_MAX_CHARGE_MSL_mA : REAL := 175000;
	CELL_CURRENT_MAX_CHARGE_RSL_mA : REAL := 175000;
	CELL_CURRENT_MAX_CHARGE_MOL_mA : REAL := 175000;
	
END_VAR

// _750_8212_PFC200/Application/CONFIG/STRING_CONFIG
{attribute 'qualified_only'}
VAR_GLOBAL CONSTANT

	BS_NR_OF_CELLS_M1 : INT := 64;
	BS_NR_OF_CELLS_M2 : INT := 64;
	BS_NR_OF_CELLS_M3 : INT := 64;
	BS_NR_OF_CELLS_M4 : INT := 16;
	BS_NR_OF_MODULES : INT := 4;
	BS_MAX_NR_OF_CELLS_PER_MODULE : INT := 64;
	BS_NR_OF_PARALLEL_CELLS : INT := 1;
	BS_TOTAL_NR_OF_CELLS : INT := BS_NR_OF_CELLS_M1 + BS_NR_OF_CELLS_M2	+ BS_NR_OF_CELLS_M3	+ BS_NR_OF_CELLS_M4;

	BS_POSITIVE_DISCHARGE_CURRENT  : BOOL := TRUE;
	BS_REST_CURRENT_mA : INT := 200;
	BS_RELAXATION_PERIOD : INT := 5000;
	
	//Value of the balancing resistors
	BS_BALANCING_RESISTANCE_ohm : INT := 100;
	
	SOC_STRING_CAPACITY_Ah : REAL := BS_NR_OF_PARALLEL_CELLS * BAT_CELL_CONFIG.CELL_NOMINAL_CAPACITY_Ah;
	SOC_STRING_CAPACITY_mAs : REAL := SOC_STRING_CAPACITY_Ah * 3600; //mAs
	SOC_STRING_CAPACITY_As : REAL := SOC_STRING_CAPACITY_mAs/1000; //mA
	
	SOC_MAXIMUM_SOC : REAL := 100;
	SOC_MINIMUM_SOC : REAL := 0;
	
END_VAR

// _750_8212_PFC200/Application/ALGO/SOC/gvSOC
{attribute 'qualified_only'}
VAR_GLOBAL
	gvSOC : typSOC;
END_VAR

// _750_8212_PFC200/Application/ALGO/SOF/gvSOF
{attribute 'qualified_only'}
VAR_GLOBAL CONSTANT
	//Maximum current in mA in charge direction that a string can sustain.
	STRING_CURRENT_CONTINUOUS_CHARGE_mA : REAL := BAT_CELL_CONFIG.CELL_CURRENT_MAX_CHARGE_MOL_mA * STRING_CONFIG.BS_NR_OF_PARALLEL_CELLS;
	
	//Maximum current in mA in discharge direction that a string can deliver.
	STRING_CURRENT_CONTINUOUS_DISCHARGE_mA : REAL := BAT_CELL_CONFIG.CELL_CURRENT_MAX_DISCHARGE_MOL_mA * STRING_CONFIG.BS_NR_OF_PARALLEL_CELLS;
	
	//Cold temperature in °C where the derating of maximum discharge current starts
	STRING_TEMPERATURE_LOW_CUTOFF_DISCHARGE_degC : REAL := BAT_CELL_CONFIG.CELL_TEMPERATURE_MIN_DISCHARGE_MOL_degC;
	
	//Cold temperature in °C where the derating of maximum discharge current is fully applied
	STRING_TEMPERATURE_LOW_LIMIT_DISCHARGE_degC : REAL := BAT_CELL_CONFIG.CELL_TEMPERATURE_MIN_DISCHARGE_MSL_degC;
	
	//Cold temperature in °C where the derating of maximum scharge current starts
	STRING_TEMPERATURE_LOW_CUTOFF_CHARGE_degC : REAL := BAT_CELL_CONFIG.CELL_TEMPERATURE_MIN_CHARGE_MOL_degC;
	
	//Cold temperature in °C where the derating of maximum scharge current is fully applied
	STRING_TEMPERATURE_LOW_LIMIT_CHARGE_degC : REAL := BAT_CELL_CONFIG.CELL_TEMPERATURE_MIN_CHARGE_MSL_degC;
	
	//Hot temperature in °C where the derating of maximum discharge current starts
	STRING_TEMPERATURE_HIGH_CUTOFF_DISCHARGE_degC : REAL := BAT_CELL_CONFIG.CELL_TEMPERATURE_MAX_DISCHARGE_MOL_degC;
	
	//Hot temperature in °C where the derating of maximum discharge current is fully applied
	STRING_TEMPERATURE_HIGH_LIMIT_DISCHARGE_degC : REAL := BAT_CELL_CONFIG.CELL_TEMPERATURE_MAX_DISCHARGE_MSL_degC;
	
	//Hot temperature in °C where the derating of maximum dcharge current starts
	STRING_TEMPERATURE_HIGH_CUTOFF_CHARGE_degC : REAL := BAT_CELL_CONFIG.CELL_TEMPERATURE_MAX_CHARGE_MOL_degC;
	
	//Hot temperature in °C where the derating of maximum charge current is fully applied
	STRING_TEMPERATURE_HIGH_LIMIT_CHARGE_degC : REAL := BAT_CELL_CONFIG.CELL_TEMPERATURE_MAX_CHARGE_MSL_degC;
	
	//Above this voltage value string should not be exposed to full current in charge direction.
	STRING_VOLTAGE_CUTOFF_CHARGE_mV : REAL := BAT_CELL_CONFIG.CELL_VOLTAGE_MAX_MOL_mV;
	
	//Above this voltage value string should not be exposed to any current in charge direction.
	STRING_VOLTAGE_LIMIT_CHARGE_mV : REAL := BAT_CELL_CONFIG.CELL_VOLTAGE_MAX_MSL_mV;
	
	//Above this voltage value string should not be exposed to full current in discharge direction.
	STRING_VOLTAGE_CUTOFF_DISCHARGE_mV : REAL := BAT_CELL_CONFIG.CELL_VOLTAGE_MIN_MOL_mV;
	
	//Above this voltage value string should not be exposed to any current in discharge direction.
	STRING_VOLTAGE_LIMIT_DISCHARGE_mV : REAL := BAT_CELL_CONFIG.CELL_VOLTAGE_MIN_MSL_mV;
	
	//Current in mA that the string should be able to discharge when in limp mode.
	STRING_CURRENT_LIMP_mA : REAL := 20000;
		
END_VAR

VAR_GLOBAL
	
	SOF_Config: typSOF_CONFIG := (
								  maximumDischargeCurrent_mA := STRING_CURRENT_CONTINUOUS_CHARGE_mA,
								  maximumDischargeCurrent_mA := STRING_CURRENT_CONTINUOUS_DISCHARGE_mA,
								  cutoffLowTemperatureDischarge_degC := STRING_TEMPERATURE_LOW_CUTOFF_DISCHARGE_degC,
								  limitLowTemperatureDischarge_degC := STRING_TEMPERATURE_LOW_LIMIT_DISCHARGE_degC,
								  cutoffLowTemperatureCharge_degC := STRING_TEMPERATURE_LOW_CUTOFF_CHARGE_degC,
								  limitLowTemperatureCharge_degC := STRING_TEMPERATURE_LOW_LIMIT_CHARGE_degC,
								  cutoffHighTemperatureDischarge_degC := STRING_TEMPERATURE_HIGH_CUTOFF_DISCHARGE_degC,
								  limitHighTemperatureDischarge_degC := STRING_TEMPERATURE_HIGH_LIMIT_DISCHARGE_degC,
								  cutoffHighTemperatureCharge_degC := STRING_TEMPERATURE_HIGH_CUTOFF_CHARGE_degC,
								  limitHighTemperatureCharge_degC := STRING_TEMPERATURE_HIGH_LIMIT_CHARGE_degC, 
								  cutoffUpperCellVoltage_mV := STRING_VOLTAGE_CUTOFF_CHARGE_mV,
								  limitUpperCellVoltage_mV := STRING_VOLTAGE_LIMIT_CHARGE_mV,
								  cutoffLowerCellVoltage_mV := STRING_VOLTAGE_CUTOFF_DISCHARGE_mV,
								  limitLowerCellVoltage_mV := STRING_VOLTAGE_LIMIT_DISCHARGE_mV,
								  limpCurrent_mA := STRING_CURRENT_LIMP_mA);

	curveRecommandedOperatingCurrent : typSOF_CURVE;							  
								  
	SOFValues : typSOF;
	
	CurrentDerating : CurrentDerating;
END_VAR

// _750_8212_PFC200/Application/CANBUS/CAN_Main
PROGRAM CAN_Main
VAR
	BMS_CAN	: CAN;	
	CAN_TX_Queue : CAN_Queue;
	CAN_TxDukosi : CAN_TxDukosi;
END_VAR


BMS_CAN.Init(IoConfig_Globals._750_658_24);

BMS_CAN.Read(CellMeas := gvCELLS.gvCellMeas, CellTemp := gvCELLS.gvCellTemp);


CAN_TxDukosi(cellControl := gvCELLS.gvCellControl,
			 ICanQueue := CAN_TX_Queue);
			 		 
BMS_CAN.Write(ICanQueue := CAN_TX_Queue);

END_PROGRAM

// _750_8212_PFC200/Application/CANBUS/CAN_TxDukosi
FUNCTION_BLOCK CAN_TxDukosi
VAR_INPUT
	cellControl : typCELL_CONTROL;
	ICanQueue : ICAN_Queue;
END_VAR
VAR_OUTPUT
END_VAR
VAR
	c : INT;
	message : typCAN_SIGNAL_TX;
	oldData : ARRAY [1..STRING_CONFIG.BS_TOTAL_NR_OF_CELLS] OF ARRAY [1..8] OF BYTE;
END_VAR


FOR c := 1 TO STRING_CONFIG.BS_TOTAL_NR_OF_CELLS DO
	
		message.Data[1] := MEM.HighByte(wValue := TO_WORD(cellControl.BAL_tgtVoltage[c]));
		message.Data[2] := MEM.LowByte(wValue := TO_WORD(cellControl.BAL_tgtVoltage[c]));
		message.Data[3] := MEM.HighByte(wValue := TO_WORD(cellControl.BAL_loadResistor[c]));
		message.Data[4] := MEM.LowByte(wValue := TO_WORD(cellControl.BAL_loadResistor[c]));
		message.Data[5] := cellControl.BAL_dutyCycle[c];
		message.Data[6] := cellControl.BAL_watchdogUnit[c];
		message.Data[7] := cellControl.BAL_watchdogCounter[c];
		message.Data[8] := cellControl.BAL_Control[c].ControlByte;
		
		IF NOT ICanQueue.isFull() THEN
			IF Compare2Arrays(message.Data, oldData[c]) THEN
				message.CAN_ID := TO_WORD(4000 + c);
				ICanQueue.addToQueue(message);
				oldData[c] := message.Data;
			END_IF
		END_IF

END_FOR

END_FUNCTION_BLOCK

// _750_8212_PFC200/Application/Utils/Compare2Arrays
FUNCTION Compare2Arrays : BOOL
VAR_INPUT
	x : ARRAY [*] OF BYTE;
	y : ARRAY [*] OF BYTE;
END_VAR
VAR
	size_x : DINT;
	start_x : DINT;
	size_y : DINT;
	start_y	 : DINT;
	diff : BYTE;
	idx : DINT;
END_VAR


size_x := UPPER_BOUND(x,1);
start_x := LOWER_BOUND(x,1);
size_y := UPPER_BOUND(y,1);
start_y := LOWER_BOUND(y,1);

Compare2Arrays := FALSE;
diff := 0;

IF size_x <> size_y THEN
	RETURN;
END_IF

FOR idx := start_x TO size_x DO
	
	diff := diff OR (x[idx] - y[idx]);

END_FOR

IF (diff <> 0) THEN
	Compare2Arrays := TRUE;
END_IF

END_FUNCTION

// _750_8212_PFC200/Application/CANBUS/Queue/ICAN_Queue
INTERFACE ICAN_Queue

METHOD addToQueue : eRET_VAL
VAR_INPUT
	item : typCAN_SIGNAL_TX;
END_VAR
END_METHOD

METHOD getFront : typCAN_SIGNAL_TX
VAR_INPUT
END_VAR
END_METHOD

METHOD isEmpty : BOOL
VAR_INPUT
END_VAR
END_METHOD

METHOD isFull : BOOL
VAR_INPUT
END_VAR
END_METHOD

METHOD removeFromQueue : eRET_VAL
VAR_INPUT
END_VAR
VAR
END_VAR
END_METHOD

END_INTERFACE

// _750_8212_PFC200/Application/CANBUS/CAN
//{attribute 'global_init_slot' := '50000'}
FUNCTION_BLOCK CAN
VAR_INPUT
END_VAR
VAR_IN_OUT
	
END_VAR
VAR_OUTPUT
END_VAR
VAR
	
	m_CAN_OpenL2 : WagoAppCanLayer2.FbCanL2Open := (udiBaudrate := 500000);
	m_CAN_CloseL2 : WagoAppCanLayer2.FbCanL2Close;
	m_CAN_ResetL2 : WagoAppCanLayer2.FbCanL2Reset;
	m_CAN_Config : WagoSysModule_75x_658.FbModuleConfigurationAndStatus;
	m_CommState : INT;
	m_Bitrate : INT;
	m_Mode : INT;
	m_29BitEnabled : BOOL;
	m_SdoEnabled : BOOL;
	m_DiagOverMbx0Enabled : BOOL;
	m_ConfigData : WagoSysModule_75x_658.WagoTypesModule_75x_658.typFullConfiguration;
	m_DiagnosisReset: BOOL;
	m_CommunicationReset : BOOL;
	I_WagoSysTypeBase : WagoAppCanLayer2.WagoTypesCan.I_WagoSysCanBase;
	I_ModuleExtended : WagoSysModule_75x_658.I_WagoModule_75x_658Extended;
	m_Init : BOOL;
	m_CAN_ReadWriteEnabled : BOOL;
	m_RX : WagoAppCanLayer2.FbCanRx29BitFrameAll;
	m_TX : WagoAppCanLayer2.FbCanTx29BitFrame;
	m_Read : BOOL;
	m_Write : BOOL;
	m_TXState : INT;
	
	//c : INT;
END_VAR
VAR_TEMP
	
END_VAR

METHOD Init
VAR_INPUT
	Port : __SYSTEM.IQueryInterface;
END_VAR
IF NOT m_Init THEN
	//Port := IoConfig_Globals._750_658_24;
	__QUERYINTERFACE(Port, I_WagoSysTypeBase);
	__QUERYINTERFACE(Port, I_ModuleExtended);
	m_Init := TRUE;
END_IF;
	
CASE m_CommState OF 
	
eCANCommState.INIT:
	m_CommState := eCANCommState.OPEN_L2;
	
eCANCommState.OPEN_L2:
	IF NOT m_CAN_OpenL2.xValid AND NOT m_CAN_OpenL2.xBusy THEN
		m_CAN_OpenL2.xEnable := TRUE;
	ELSIF m_CAN_OpenL2.xValid AND NOT m_CAN_OpenL2.xError THEN
		m_CAN_ReadWriteEnabled := TRUE;
	ELSIF m_CAN_OpenL2.xError THEN
		m_CAN_ReadWriteEnabled := FALSE;
		m_CAN_OpenL2.xEnable := FALSE;	
		m_CommState := eCANCommState.CLOSE_L2;
	END_IF;	

eCANCommState.CLOSE_L2:
	m_CAN_CloseL2.xExecute := TRUE;
	IF m_CAN_CloseL2.xDone THEN
		m_CommState := eCANCommState.RESET_L2;
		m_CAN_CloseL2.xExecute := FALSE;
	END_IF
	
eCANCommState.RESET_L2:	
	m_CAN_ResetL2.xExecute := TRUE;
	IF m_CAN_ResetL2.xDone THEN
		m_CommState := eCANCommState.OPEN_L2;
		m_CAN_ResetL2.xExecute := FALSE;
	END_IF

eCANCommState.CONFIG_L2:
	m_Bitrate := 5;
	m_Mode := 1;
	m_29BitEnabled := TRUE;
	m_SdoEnabled := FALSE;
	m_DiagOverMbx0Enabled := TRUE;

	IF NOT m_CAN_Config.xBusy AND NOT m_CAN_Config.xDone THEN
		m_CAN_Config.xExecute := TRUE;
		m_CAN_Config.xWriteRead := TRUE;
		m_CAN_Config.xSaveValues := TRUE;
	ELSIF NOT m_CAN_Config.xBusy AND m_CAN_Config.xDone	THEN
		m_CAN_Config.xExecute := FALSE;
		m_CAN_Config.xWriteRead := FALSE;
		m_CAN_Config.xSaveValues := FALSE;
		m_CommState := eCANCommState.READ;
	END_IF
	
END_CASE

m_CAN_OpenL2(I_Port := I_WagoSysTypeBase,
			 udiBaudrate := 500000);

m_CAN_CloseL2(
	I_Port:= I_WagoSysTypeBase);			 

m_CAN_ResetL2(
	I_Port:= I_WagoSysTypeBase);
			 
m_CAN_Config(
	I_Port:= I_ModuleExtended, 
	eBitrate:= m_Bitrate, 
	eMode:= m_Mode, 
	x29BitEnabled:= m_29BitEnabled, 
	xSdoEnabled:= m_SdoEnabled, 
	xDiagOverMbx0Enabled:= m_DiagOverMbx0Enabled, 
	typConfigData:= m_ConfigData, 
	xDiagnosisReset:= m_DiagnosisReset, 
	xCommunicationReset:= m_CommunicationReset);
END_METHOD

METHOD Read
VAR_INPUT 
	CellMeas : REFERENCE TO typCELL_MEAS;
	CellTemp : REFERENCE TO typCELL_TEMP;
END_VAR

VAR
	_idx : INT;
END_VAR

GVL_CAN_Data.arrCANDataRX[1].Info.TimeOutDelay(	IN := TRUE,
					   							PT := CAN_CONFIG.CAN_TIMEOUT_DELAY,
					   							Q => GVL_CAN_Data.arrCANDataRX[1].Info.TimeOutAlarm);	 

m_RX(xEnable := m_CAN_ReadWriteEnabled,
	 I_Port := I_WagoSysTypeBase,
	 xRxTrigger := m_Read);

IF NOT m_Read THEN
	m_Read := TRUE;
END_IF
							 
// GVL_CAN_Data.arrCANDataRX[1].Info.Timpstamp := T_PLC_MS();										 
// //IF m_pktCounter <> m_oldPktCounter THEN
// 	IF GVL_CAN_Data.arrCANDataRX[1].Config.ID = m_RX.dwRxId + CAN_CONFIG.CAN_OFFSET THEN
// 			GVL_CAN_Data.arrCANDataRX[1].Info.TimeOutDelay(IN := FALSE);
// 			GVL_CAN_Data.arrCANDataRX[1].Info.Data := m_RX.aRxBuffer;
// 			GVL_CAN_Data.arrCANDataRX[1].Info.pktReceived := m_RX.bRxNBytes;// + Data.Info.pktReceived;	
// 			GVL_CAN_Data.arrCANDataRX[1].Info.deltaT := GVL_CAN_Data.arrCANDataRX[1].Info.Timpstamp - GVL_CAN_Data.arrCANDataRX[1].Info.previousTimestamp;
// 			GVL_CAN_Data.arrCANDataRX[1].Info.previousTimestamp := GVL_CAN_Data.arrCANDataRX[1].Info.Timpstamp;
// 			GVL_CAN_Data.arrCANDataRX[1].Info.pktCounter_old := GVL_CAN_Data.arrCANDataRX[1].Info.pktReceived;
// 	END_IF
	
UpdateCellData(m_RX.dwRxId, m_Rx.aRxBuffer, CellMeas, CellTemp);	


//END_IF
END_METHOD

METHOD PRIVATE UpdateCellData
VAR_INPUT
	CanID : DWORD;
	CanMessage : ARRAY [1..8] OF BYTE;
	CellMeas : REFERENCE TO typCELL_MEAS;
	CellTemp : REFERENCE TO typCELL_TEMP;
END_VAR
VAR
	_DecodedCAN : typCAN_ID;
	_CellIdx : INT;
END_VAR

_DecodedCAN := DecodeCAN_ID(CanID);
_CellIdx := TO_INT(STRING_CONFIG.BS_MAX_NR_OF_CELLS_PER_MODULE * (_DecodedCAN.SA - 1) + _DecodedCAN.CA);


CASE _DecodedCAN.ID OF
	
	eCAN_MESSAGE_ID.CELL_MEAS:
		CellMeas.voltage.cellVoltage_mV[_CellIdx] := CAN_TO_INT(StartByte := 1, Data := ADR(CanMessage));
		CellMeas.balCurrent.cellBalCurrent_mAmps[_CellIdx] := CAN_TO_INT(StartByte := 3, Data := ADR(CanMessage));
		CellMeas.cellStatus[_CellIdx].AlarmWord := TO_WORD(CAN_TO_INT(StartByte := 5, Data := ADR(CanMessage)));
		CellMeas.cellBalStatus[_CellIdx].StatusWord := TO_WORD(CAN_TO_INT(StartByte := 7, Data := ADR(CanMessage)));
		CellMeas.timeStamp[_CellIdx] := T_PLC_MS();
		CellMeas.previousTimeStamp[_CellIdx] := CellMeas.timeStamp[_CellIdx];
	
	eCAN_MESSAGE_ID.CELL_TEMP:
		CellTemp.temperature.cellTemperature_deg[_CellIdx] := CAN_TO_INT(StartByte := 1, Data := ADR(CanMessage));	
		CellTemp.DyeTemperature.cellDyeTemperature_deg[_CellIdx] := CAN_TO_INT(StartByte := 3, Data := ADR(CanMessage));	
		CellTemp.timeStamp[_CellIdx] := T_PLC_MS();
		CellTemp.previousTimeStamp[_CellIdx] := CellTemp.timeStamp[_CellIdx];
END_CASE
END_METHOD

METHOD Write
VAR_INPUT
	ICanQueue : ICAN_Queue;
END_VAR
VAR
	canRxSignal : typCAN_SIGNAL_TX;
END_VAR

IF ICanQueue.isEmpty() THEN
	RETURN;
END_IF 

CASE m_TXState OF
	
	eTX_STATUS.ST_CAN_TX_INIT:
		IF m_CAN_ReadWriteEnabled THEN
			m_TXState := eTX_STATUS.ST_CAN_TX_NEXT_REQ;
		END_IF

	eTX_STATUS.ST_CAN_TX_NEXT_REQ:

		canRxSignal := ICanQueue.getFront();
		m_TXState := eTX_STATUS.ST_CAN_TX_WRITE;
		m_Write := TRUE;
		
	eTX_STATUS.ST_CAN_TX_WRITE:
		IF NOT m_Write AND NOT m_TX.xError AND m_TX.xValid THEN
			m_TXState := eTX_STATUS.ST_CAN_TX_NEXT_REQ;	
			ICanQueue.removeFromQueue();
		END_IF
		
END_CASE



m_TX(xEnable := m_CAN_ReadWriteEnabled,
	 xTxTrigger := m_Write,
	 I_Port := I_WagoSysTypeBase,
	 dwCanId := canRxSignal.CAN_ID,
	 aTxBuffer := canRxSignal.Data,
	 bTxNBytes := 8);
END_METHOD

END_FUNCTION_BLOCK

// _750_8212_PFC200/Application/Utils/T_PLC_MS
FUNCTION T_PLC_MS : DWORD
VAR CONSTANT
	debug : BOOL := 0;
	N : INT := 0;
	offset : DWORD := 0;
END_VAR
VAR
	tx : TIME;
END_VAR

(*
version 1.2	16. nov 2008
programmer 	hugo
tested by	oscat

T_PLC_MS reads the internal PLC timer and return the time, it has the advantage to be able to set a debug mode 
and speed up the counter to test the plc timer overrun which occurs every 50 days respectively 25 days at siemens S7
this routine also allows to correct the behavior of s7 where the internal plc counter will not count all 32 bits.

*)

tx := TIME();
T_PLC_MS := TIME_TO_DWORD(Tx);

IF debug THEN
	T_PLC_MS := (SHL(T_PLC_MS,N) OR SHL(DWORD#1,N)-1) + OFFSET;
END_IF;

END_FUNCTION

// _750_8212_PFC200/Application/BMSUtils/DecodeCAN_ID
FUNCTION DecodeCAN_ID : typCAN_ID
VAR_INPUT
	CAN_ID : DWORD;
END_VAR
VAR
	_dwPGN : DWORD;
END_VAR

// 
// DecodeCAN_ID.SA := DWORD_TO_BYTE(SHR(CAN_ID,SHL(0,3)));
// _dwPGN := SHL(CAN_ID, 8);
// _dwPGN := SHR(_dwPGN, 8);
// _dwPGN := SHR(_dwPGN, 8);
// DecodeCAN_ID.PGN := TO_WORD(_dwPGN);
// DecodeCAN_ID.P := DWORD_TO_BYTE(SHR(CAN_ID,SHL(3,3)));

DecodeCAN_ID.SA := BYTE_OF_DWORD(CAN_ID, 0);
DecodeCAN_ID.CA := BYTE_OF_DWORD(CAN_ID, 1);
DecodeCAN_ID.ID := BYTE_OF_DWORD(CAN_ID, 2);
DecodeCAN_ID.P := BYTE_OF_DWORD(CAN_ID, 3);

END_FUNCTION

// _750_8212_PFC200/Application/Utils/BYTE_OF_DWORD
FUNCTION BYTE_OF_DWORD : BYTE
VAR_INPUT
	in : DWORD;
	N : BYTE;
END_VAR


(*
version 1.2	30. oct. 2008
programmer 	hugo
tested by	oscat

this function extracts a single byte from the nth position from right (right is lowest byte) 
the lower byte (starting with Bit0 from in) is selected with N=0.
*)

BYTE_OF_DWORD := DWORD_TO_BYTE(SHR(in,SHL(n,3)));

(* revision history
hm	17. jan 2007	rev 1.0
	original version

hm	2. jan 2008		rev 1.1
	improved performance

hm	30. oct. 2008	rev 1.2
	improved performance
*)

END_FUNCTION

// _750_8212_PFC200/Application/CANBUS/CANUtils/CAN_TO_INT
FUNCTION CAN_TO_INT : INT
VAR_INPUT
	StartByte : INT;
	Data : POINTER TO ARRAY[1..8] OF BYTE;
END_VAR
VAR
	b0 : BYTE;
    b1 : BYTE;
END_VAR

IF (Data = 0) THEN RETURN; END_IF;

b0 := Data^[StartByte];
b1 := Data^[StartByte+1];

CAN_TO_INT := TO_INT(SHL(BYTE_TO_WORD(b1),8) OR BYTE_TO_WORD(B0));

END_FUNCTION

// _750_8212_PFC200/Application/CANBUS/Queue/CAN_Queue
FUNCTION_BLOCK CAN_Queue IMPLEMENTS ICAN_Queue
VAR_INPUT
END_VAR
VAR_OUTPUT
END_VAR
VAR
	buffer : ARRAY[0..MAX_ELEMENTS-1] OF typCAN_SIGNAL_TX;
	front : INT := -1;
	rear : INT := -1;
	size : INT := MAX_ELEMENTS;
	stop: INT;
	test: INT;
END_VAR
VAR CONSTANT
	MAX_ELEMENTS : INT := 50;
END_VAR

METHOD addToQueue : eRET_VAL
VAR_INPUT
	item : typCAN_SIGNAL_TX;
END_VAR

VAR
	
END_VAR
addToQueue := eRET_VAL.STD_NOT_OK;
IF (isFull()) THEN
	RETURN;
ELSIF (front = -1) THEN
	front := rear := 0;
	buffer[rear] := item;
ELSIF (rear = size - 1 AND front <> 0) THEN
	rear := 0;
	buffer[rear] := item;
ELSE
	rear := rear + 1;
	buffer[rear] := item;
END_IF

addToQueue := eRET_VAL.STD_OK;
END_METHOD

METHOD getFront : typCAN_SIGNAL_TX
VAR_INPUT
END_VAR
IF isEmpty() THEN
	RETURN;
END_IF
IF (front = -1) THEN
	front := 0;
END_IF

getFront := buffer[front];
END_METHOD

METHOD isEmpty : BOOL
VAR_INPUT
END_VAR
isEmpty := (front = -1);
END_METHOD

METHOD isFull : BOOL
VAR_INPUT
END_VAR
isFull := (((front = 0) AND (rear = size - 1)) OR ((rear + 1) MOD size = front));
END_METHOD

METHOD removeFromQueue : eRET_VAL
VAR_INPUT
END_VAR
VAR
	elem : typCAN_SIGNAL_TX;
END_VAR
removeFromQueue := eRET_VAL.STD_NOT_OK;
IF (isEmpty()) THEN
	RETURN;
END_IF

elem := buffer[front];
IF (front = rear) THEN
	front := -1;
	rear := -1;
ELSIF (front = size - 1) THEN
	front := 0;
ELSE 
	front := front + 1;
END_IF

removeFromQueue := eRET_VAL.STD_OK;
END_METHOD

END_FUNCTION_BLOCK

// _750_8212_PFC200/Application/Simulate
PROGRAM Simulate
VAR
	c : INT;
	simVoltage : BOOL;
END_VAR

IF simVoltage THEN
	
	FOR c := 1 TO STRING_CONFIG.BS_TOTAL_NR_OF_CELLS DO
		gvCELLS.gvCellMeas.voltage.cellVoltage_mV[c] := 2000;
	END_FOR
	simVoltage := FALSE;
END_IF

END_PROGRAM

// _750_8212_PFC200/Application/Main
PROGRAM Main
VAR
xInit : BOOL;

END_VAR


IF xInit THEN
	gvBMS.BalancingControl.SetStateRequest(stateRequest := eBAL_STATE_REQUEST.BAL_STATE_ALLOWBALANCING_REQUEST);
	gvBMS.BalancingControl.SetStateRequest(stateRequest := eBAL_STATE_REQUEST.BAL_STATE_GLOBAL_ENABLE_REQUEST);
ELSE
	gvBMS.BalancingControl.SetStateRequest(stateRequest := eBAL_STATE_REQUEST.BAL_STATE_GLOBAL_DISABLE_REQUEST);
	gvBMS.BalancingControl.SetStateRequest(stateRequest := eBAL_STATE_REQUEST.BAL_STATE_GLOBAL_DISABLE_REQUEST);
END_IF

gvBMS.StringStat.Main();
gvSOF.CurrentDerating.Calculate();
gvBMS.BalancingControl.Run();
gvBMS.Pulse1Sec();

END_PROGRAM

// _750_8212_PFC200/Application/BALANCING/BalancingControl
FUNCTION_BLOCK BalancingControl
VAR_INPUT
	cellVoltage : REFERENCE TO typCELL_VOLTAGE;
	minMax : REFERENCE TO typMIN_MAX;
	balControl : REFERENCE TO typBALANCING_CONTROL;
END_VAR
VAR_OUTPUT
END_VAR
VAR
	bal_State : typBAL_STATE;
END_VAR

METHOD Activate : BOOL
VAR_INPUT

END_VAR
VAR
	cellBalancingCurrent : REAL;
	difference : INT;
	nrBalancedCells : INT;
	c : INT;
	finished : BOOL;
	minVoltage : REAL;
END_VAR

finished := TRUE;
minVoltage := minMax.minimumCellVoltage_mV;

FOR c := 1 TO STRING_CONFIG.BS_TOTAL_NR_OF_CELLS DO
	IF cellVoltage.cellVoltage_mV[c] > (minVoltage + bal_State.balancingThreshold) THEN
		balControl.balancingState[c] := 1;
		finished := FALSE;
		bal_State.balancingThreshold := balControl.threshold_mV;
		bal_state.active := TRUE;
		balControl.enableBalancing := TRUE;
		nrBalancedCells := nrBalancedCells + 1;
	ELSE
		balControl.balancingState[c] := 0;
	END_IF
END_FOR

balControl.nrBalancedCells := nrBalancedCells;

Activate := finished;
END_METHOD

METHOD CheckStateRequest : eBAL_RETURN
VAR_INPUT
	CurrentState : REFERENCE TO typBAL_STATE;
	stateRequest : eBAL_STATE_REQUEST;
END_VAR
IF (stateRequest = eBAL_STATE_REQUEST.BAL_STATE_ERROR_REQUEST) THEN
	CheckStateRequest := eBAL_RETURN.BAL_OK;
	RETURN;
END_IF

IF (stateRequest = eBAL_STATE_REQUEST.BAL_STATE_GLOBAL_ENABLE_REQUEST) THEN
	CurrentState.balancingGlobalAllowed := TRUE;
	CheckStateRequest := eBAL_RETURN.BAL_OK;
	RETURN;
END_IF

IF (stateRequest = eBAL_STATE_REQUEST.BAL_STATE_GLOBAL_DISABLE_REQUEST) THEN
	CurrentState.balancingGlobalAllowed := FALSE;
	CheckStateRequest := eBAL_RETURN.BAL_OK;
	RETURN;
END_IF

IF (stateRequest = eBAL_STATE_REQUEST.BAL_STATE_NO_BALANCING_REQUEST) OR (stateRequest = eBAL_STATE_REQUEST.BAL_STATE_ALLOWBALANCING_REQUEST) THEN
	CheckStateRequest := eBAL_RETURN.BAL_OK;
	RETURN;
END_IF

IF (CurrentState.stateRequest = eBAL_STATE_REQUEST.BAL_STATE_NO_REQUEST) THEN
	IF (stateRequest = eBAL_STATE_REQUEST.BAL_STATE_INIT_REQUEST) THEN
		IF (CurrentState.state = eBAL_STATE.BAL_STATEMACH_UNINITIALIZED) THEN
			CheckStateRequest := eBAL_RETURN.BAL_OK;
			RETURN;
		ELSE
			CheckStateRequest := eBAL_RETURN.BAL_ALREADY_INITIALIZED;
			RETURN;
		END_IF
	ELSE
		CheckStateRequest := eBAL_RETURN.BAL_ILLEGAL_REQUEST;
		RETURN;
	END_IF
ELSE
	CheckStateRequest := eBAL_RETURN.BAL_REQUEST_PENDING;
	RETURN;
END_IF
END_METHOD

METHOD Deactivate
VAR_INPUT
END_VAR
VAR
	idx : INT;
END_VAR

FOR idx := 1 TO STRING_CONFIG.BS_TOTAL_NR_OF_CELLS DO
	balControl.balancingState[idx] := 0;
END_FOR
balControl.nrBalancedCells := 0;
balControl.enableBalancing := 0;
bal_State.active := FALSE;
END_METHOD

METHOD Process
VAR_INPUT
	Activate : BOOL;
END_VAR
END_METHOD

METHOD ProcessState_Balancing
VAR_INPUT
	stateRequest : eBAL_STATE_REQUEST;
END_VAR
IF (stateRequest = eBAL_STATE_REQUEST.BAL_STATE_NO_BALANCING_REQUEST) THEN
	bal_State.balancingAllowed := FALSE;
END_IF

IF (stateRequest = eBAL_STATE_REQUEST.BAL_STATE_ALLOWBALANCING_REQUEST) THEN
	bal_State.balancingAllowed := TRUE;
END_IF

IF (bal_State.balancingGlobalAllowed = FALSE) THEN
	IF (bal_State.active) THEN
		Deactivate();
	END_IF
	bal_State.active := FALSE;
	bal_State.state := eBAL_STATE.BAL_STATEMACH_BALANCE;
	bal_State.substate := eBAL_SUB_STATE.BAL_ENTRY;
	RETURN;
END_IF

IF (bal_State.substate = eBAL_SUB_STATE.BAL_ENTRY) THEN
	IF (bal_State.balancingGlobalAllowed = FALSE) THEN
		IF (bal_State.active) THEN
			Deactivate();
		END_IF
		bal_State.active := FALSE;
		bal_State.state := eBAL_STATE.BAL_STATEMACH_BALANCE;
		bal_State.substate := eBAL_SUB_STATE.BAL_ENTRY;
	ELSE
		bal_State.substate := eBAL_SUB_STATE.BAL_CHECK_LOWEST_VOLTAGE;
	END_IF
ELSIF (bal_State.substate = eBAL_SUB_STATE.BAL_CHECK_LOWEST_VOLTAGE) THEN
	bal_State.substate := eBAL_SUB_STATE.BAL_CHECK_CURRENT;
	IF (minMax.minimumCellVoltage_mV <= BALANCING_CONFIG.BAL_LOWER_VOLTAGE_LIMIT_mV) OR 
	    (minMax.maximumTemperature_degC >= BALANCING_CONFIG.BAL_UPPER_TEMPERATURE_LIMIT_degC) THEN
		IF (bal_State.active) THEN
			Deactivate();
		END_IF
		bal_State.active := FALSE;
		bal_State := eBAL_STATE.BAL_STATEMACH_CHECK_BALANCING;
		bal_State.substate := eBAL_SUB_STATE.BAL_ENTRY;
	END_IF
	RETURN;
ELSIF (bal_State.substate = eBAL_SUB_STATE.BAL_CHECK_CURRENT) THEN
	IF (gvBMS.Fb_String.GetStringState() = eBMS_CURRENT_FLOW_STATE.AT_REST) THEN
		bal_State.substate := eBAL_SUB_STATE.BAL_ACTIVATE_BALANCING;
	ELSE
		IF (bal_State.active) THEN
			Deactivate();
		END_IF
		bal_State.active := FALSE;
		bal_State := eBAL_STATE.BAL_STATEMACH_CHECK_BALANCING;
		bal_State.substate := eBAL_SUB_STATE.BAL_ENTRY;	
	END_IF
	RETURN;
ELSIF (bal_State.substate = eBAL_SUB_STATE.BAL_ACTIVATE_BALANCING) THEN
	IF (bal_State.balancingGlobalAllowed = FALSE) THEN
		IF (bal_State.active) THEN
			Deactivate();
		END_IF
		bal_State.active := FALSE;
		bal_State.state := eBAL_STATE.BAL_STATEMACH_BALANCE;
		bal_State.substate := eBAL_SUB_STATE.BAL_ENTRY;
	ELSE
		IF (Activate() = TRUE) THEN
			bal_State.balancingThreshold := balControl.threshold_mV + BALANCING_CONFIG.BAL_HYSTERESIS_mV;
			bal_State.state := eBAL_STATE.BAL_STATEMACH_CHECK_BALANCING;
			bal_State.substate := eBAL_SUB_STATE.BAL_ENTRY;
		ELSE
			bal_State.state := eBAL_STATE.BAL_STATEMACH_BALANCE;
			bal_State.substate := eBAL_SUB_STATE.BAL_ENTRY;
		END_IF
	END_IF
	RETURN;
END_IF
END_METHOD

METHOD ProcessState_CheckBalancing
VAR_INPUT
	stateRequest : eBAL_STATE_REQUEST;
END_VAR
IF (stateRequest = eBAL_STATE_REQUEST.BAL_STATE_NO_BALANCING_REQUEST) THEN
	bal_State.balancingAllowed := FALSE;
END_IF

IF (stateRequest = eBAL_STATE_REQUEST.BAL_STATE_ALLOWBALANCING_REQUEST) THEN
	bal_State.balancingAllowed := TRUE;
END_IF

IF ((bal_State.balancingAllowed = FALSE) OR (bal_State.balancingGlobalAllowed = FALSE)) THEN
	Deactivate();
	bal_State.active := FALSE;
ELSE
	IF (gvBMS.Fb_String.GetStringState() = eBMS_CURRENT_FLOW_STATE.AT_REST) THEN
		bal_State.state := eBAL_STATE.BAL_STATEMACH_BALANCE;
		bal_State.substate := eBAL_SUB_STATE.BAL_ENTRY;
	END_IF
END_IF
END_METHOD

METHOD SetStateRequest : eBAL_RETURN
VAR_INPUT
	stateRequest : eBAL_STATE_REQUEST;
END_VAR
VAR
	retVal : eBAL_RETURN;
END_VAR
SetStateRequest := eBAL_RETURN.BAL_OK;

retVal := CheckStateRequest(bal_State, stateRequest);

IF retVal = eBAL_RETURN.BAL_OK THEN
	bal_State.stateRequest := stateRequest;
END_IF

SetStateRequest := retVal;
END_METHOD

END_FUNCTION_BLOCK

// _750_8212_PFC200/Application/ALGO/SOF/CurrentDerating
FUNCTION_BLOCK CurrentDerating
VAR_INPUT
END_VAR
VAR_OUTPUT
END_VAR
VAR
END_VAR

METHOD Calculate
VAR_INPUT
END_VAR
VAR
	allowedCurrent : typSOF_CURRENT_LIMITS;
	voltageBasedSof : typSOF_CURRENT_LIMITS;
	temperatureBasedSof : typSOF_CURRENT_LIMITS;
	minCharge : REAL;
	minDischarge : REAL;
END_VAR
//IF BMS_IsConnected() then
	CalculateVoltageBasedCurrentLimits(minCellVoltage := gvBMS.gvMinMax.minimumCellVoltage_mV,
									   maxCellVoltage := gvBMS.gvMinMax.maximumCellVoltage_mV,
									   AllowedVoltageBasedCurrent := voltageBasedSof,
									   CalculatedCurveValues := gvSOF.curveRecommandedOperatingCurrent,
									   ConfigurationValues := gvSOF.SOF_Config);
									   
	CalculateTemperatureBasedCurrentLimit(minCellTemperature := gvBMS.gvMinMax.minimumTemperature_degC,
										  maxCellTemperature := gvBMS.gvMinMax.maximumTemperature_degC,
										  AllowedTemperatureBasedCurrent := temperatureBasedSof,
										  CalculatedCurveValues := gvSOF.curveRecommandedOperatingCurrent,
										  ConfigurationValues := gvSOF.SOF_Config);	

	allowedCurrent.ContinuosChargeCurrent := MIN(voltageBasedSof.ContinuosChargeCurrent, temperatureBasedSof.ContinuosChargeCurrent);
	allowedCurrent.PeakChargeCurrent := MIN(voltageBasedSof.PeakChargeCurrent, temperatureBasedSof.PeakChargeCurrent);
	allowedCurrent.ContinuosDischargeCurrent := MIN(voltageBasedSof.ContinuosDischargeCurrent, temperatureBasedSof.ContinuosDischargeCurrent);
	allowedCurrent.PeakDischargeCurrent := MIN(voltageBasedSof.PeakDischargeCurrent, temperatureBasedSof.PeakDischargeCurrent);
	
	gvSOF.SOFValues.recommandedContinuosChargeCurrent := allowedCurrent.ContinuosChargeCurrent;
	gvSOF.SOFValues.recommandedContinuosDischargeCurrent := allowedCurrent.ContinuosDischargeCurrent;
	gvSOF.SOFValues.recommandedPeakChargeCurrent := allowedCurrent.PeakChargeCurrent;
	gvSOF.SOFValues.recommandedPeakDischargeCurrent := allowedCurrent.PeakDischargeCurrent;
	
	gvSOF.SOFValues.recommandedContinuosChargeCurrent := allowedCurrent.ContinuosChargeCurrent;
	gvSOF.SOFValues.recommandedContinuosDischargeCurrent := allowedCurrent.ContinuosDischargeCurrent;
	gvSOF.SOFValues.recommandedPeakChargeCurrent := allowedCurrent.PeakChargeCurrent;
	gvSOF.SOFValues.recommandedPeakDischargeCurrent := allowedCurrent.PeakDischargeCurrent;
	
//else
// 	gvSOF.SOFValues.recommandedContinuosChargeCurrent := 0;
// 	gvSOF.SOFValues.recommandedContinuosDischargeCurrent := 0;
// 	gvSOF.SOFValues.recommandedPeakChargeCurrent := 0;
// 	gvSOF.SOFValues.recommandedPeakDischargeCurrent := 0;	
//end_if

// IF (BMS_IsTransitionToErrorStateActive() = TRUE) THEN
// 	sof_tableSofValues.recommendedContinuousPackChargeCurrent_mA    = 0.0f;
// 	sof_tableSofValues.recommendedContinuousPackDischargeCurrent_mA = 0.0f;
// 	sof_tableSofValues.recommendedPeakPackChargeCurrent_mA          = 0.0f;
// 	sof_tableSofValues.recommendedPeakPackDischargeCurrent_mA       = 0.0f;
// END_IF
END_METHOD

METHOD PRIVATE CalculateCurves
VAR_INPUT
	CalculatedCurveValues : REFERENCE TO typSOF_CURVE;
	ConfigurationValues : REFERENCE TO typSOF_CONFIG;
END_VAR
CalculatedCurveValues.slopeLowTemperatureDischarge := (ConfigurationValues.maximumDischargeCurrent_mA - ConfigurationValues.limpCurrent_mA) / 
													  (ConfigurationValues.cutoffLowTemperatureDischarge_degC - ConfigurationValues.limitLowTemperatureDischarge_degC);
													 
CalculatedCurveValues.offsetLowTemperatureDischarge := ConfigurationValues.limpCurrent_mA - (CalculatedCurveValues.slopeLowTemperatureDischarge - ConfigurationValues.limitLowTemperatureDischarge_degC);

CalculatedCurveValues.slopeHighTemperatureDischarge := (0 - ConfigurationValues.maximumDischargeCurrent_mA) / 
													   (ConfigurationValues.limitHighTemperatureDischarge_degC - ConfigurationValues.cutoffHighTemperatureDischarge_degC);
													  
CalculatedCurveValues.offsetHighTemperatureDischarge := 0 - (CalculatedCurveValues.slopeHighTemperatureDischarge - ConfigurationValues.limitHighTemperatureDischarge_degC);													  
													  
CalculatedCurveValues.slopeLowTemperatureCharge := (ConfigurationValues.maximumChargeCurrent_mA - 0) / 
												   (ConfigurationValues.cutoffLowTemperatureCharge_degC - ConfigurationValues.limitLowTemperatureCharge_degC);
													 
CalculatedCurveValues.offsetLowTemperatureCharge := 0 - (CalculatedCurveValues.slopeLowTemperatureCharge - ConfigurationValues.limitLowTemperatureCharge_degC);

CalculatedCurveValues.slopeHighTemperatureCharge := (0 - ConfigurationValues.maximumChargeCurrent_mA) / 
												    (ConfigurationValues.limitHighTemperatureCharge_degC - ConfigurationValues.cutoffHighTemperatureCharge_degC);
													 
CalculatedCurveValues.offsetHighTemperatureDischarge := 0 - (CalculatedCurveValues.slopeHighTemperatureCharge - ConfigurationValues.limitHighTemperatureCharge_degC);				

CalculatedCurveValues.slopeUpperCellVoltage := (ConfigurationValues.maximumDischargeCurrent_mA - 0) / 
											   (ConfigurationValues.cutoffLowerCellVoltage_mV - ConfigurationValues.limitLowerCellVoltage_mV); 
											   
CalculatedCurveValues.offsetUpperCellVoltage := 0 - (CalculatedCurveValues.slopeUpperCellVoltage - ConfigurationValues.limitLowerCellVoltage_mV);

CalculatedCurveValues.slopeLowerCellVoltage := (ConfigurationValues.maximumChargeCurrent_mA - 0) / 
											   (ConfigurationValues.cutoffUpperCellVoltage_mV - ConfigurationValues.limitUpperCellVoltage_mV);
											   
CalculatedCurveValues.offsetLowerCellVoltage := 0 - (CalculatedCurveValues.slopeLowerCellVoltage - ConfigurationValues.limitLowerCellVoltage_mV);
END_METHOD

METHOD PRIVATE CalculateTemperatureBasedCurrentLimit
VAR_INPUT
	minCellTemperature : REAL;
	maxCellTemperature : REAL;
	AllowedTemperatureBasedCurrent : REFERENCE TO typSOF_CURRENT_LIMITS;
	CalculatedCurveValues : REFERENCE TO typSOF_CURVE;
	ConfigurationValues : REFERENCE TO typSOF_CONFIG;
END_VAR
VAR
	tempCurrentLimits : typSOF_CURRENT_LIMITS;
END_VAR
IF (minCellTemperature <= ConfigurationValues.limitLowTemperatureDischarge_degC) THEN
	AllowedTemperatureBasedCurrent.ContinuosDischargeCurrent := ConfigurationValues.limpCurrent_mA;
	AllowedTemperatureBasedCurrent.PeakDischargeCurrent := ConfigurationValues.limpCurrent_mA;
ELSE
	IF (minCellTemperature <= ConfigurationValues.cutoffLowTemperatureDischarge_degC) THEN
		AllowedTemperatureBasedCurrent.ContinuosDischargeCurrent := (CalculatedCurveValues.slopeLowTemperatureDischarge*minCellTemperature) + CalculatedCurveValues.offsetLowTemperatureDischarge;
		AllowedTemperatureBasedCurrent.PeakDischargeCurrent := AllowedTemperatureBasedCurrent.ContinuosDischargeCurrent;
	ELSE
		AllowedTemperatureBasedCurrent.ContinuosDischargeCurrent := ConfigurationValues.maximumDischargeCurrent_mA;
		AllowedTemperatureBasedCurrent.PeakDischargeCurrent := ConfigurationValues.maximumDischargeCurrent_mA;	
	END_IF
END_IF

IF (minCellTemperature <= ConfigurationValues.limitLowTemperatureCharge_degC) THEN
	AllowedTemperatureBasedCurrent.ContinuosDischargeCurrent := 0;
	AllowedTemperatureBasedCurrent.PeakDischargeCurrent := 0;
ELSE
	IF (minCellTemperature <= ConfigurationValues.cutoffLowTemperatureCharge_degC) THEN
		AllowedTemperatureBasedCurrent.ContinuosDischargeCurrent := (CalculatedCurveValues.slopeLowTemperatureCharge*minCellTemperature) + CalculatedCurveValues.offsetLowTemperatureCharge;
		AllowedTemperatureBasedCurrent.PeakChargeCurrent := AllowedTemperatureBasedCurrent.ContinuosChargeCurrent;
	ELSE
		AllowedTemperatureBasedCurrent.ContinuosChargeCurrent := ConfigurationValues.maximumChargeCurrent_mA;
		AllowedTemperatureBasedCurrent.PeakDischargeCurrent := ConfigurationValues.maximumChargeCurrent_mA;	
	END_IF
END_IF

IF (maxCellTemperature >= ConfigurationValues.limitHighTemperatureDischarge_degC) THEN
	AllowedTemperatureBasedCurrent.ContinuosDischargeCurrent := 0;
	AllowedTemperatureBasedCurrent.PeakDischargeCurrent := 0;
ELSE
	IF (maxCellTemperature >= ConfigurationValues.cutoffHighTemperatureDischarge_degC) THEN
		tempCurrentLimits.ContinuosDischargeCurrent := (CalculatedCurveValues.slopeHighTemperatureDischarge*maxCellTemperature) + CalculatedCurveValues.offsetHighTemperatureDischarge;
		tempCurrentLimits.PeakDischargeCurrent := tempCurrentLimits.ContinuosDischargeCurrent;
	ELSE
		tempCurrentLimits.ContinuosDischargeCurrent := ConfigurationValues.maximumDischargeCurrent_mA;
		tempCurrentLimits.PeakDischargeCurrent := ConfigurationValues.maximumDischargeCurrent_mA;	
	END_IF
	AllowedTemperatureBasedCurrent.ContinuosDischargeCurrent := MIN(AllowedTemperatureBasedCurrent.ContinuosDischargeCurrent, tempCurrentLimits.ContinuosDischargeCurrent);
	AllowedTemperatureBasedCurrent.ContinuosDischargeCurrent := MIN(AllowedTemperatureBasedCurrent.PeakDischargeCurrent, tempCurrentLimits.PeakDischargeCurrent);
END_IF

IF (maxCellTemperature >= ConfigurationValues.limitHighTemperatureCharge_degC) THEN
	AllowedTemperatureBasedCurrent.ContinuosChargeCurrent := 0;
	AllowedTemperatureBasedCurrent.PeakChargeCurrent := 0;
ELSE
	IF (maxCellTemperature >= ConfigurationValues.cutoffHighTemperatureCharge_degC) THEN
		tempCurrentLimits.ContinuosChargeCurrent := (CalculatedCurveValues.slopeHighTemperatureCharge*maxCellTemperature) + CalculatedCurveValues.offsetHighTemperatureCharge;
		tempCurrentLimits.PeakChargeCurrent := tempCurrentLimits.ContinuosChargeCurrent;
	ELSE
		tempCurrentLimits.ContinuosChargeCurrent := ConfigurationValues.maximumChargeCurrent_mA;
		tempCurrentLimits.PeakChargeCurrent := ConfigurationValues.maximumChargeCurrent_mA;	
	END_IF
	AllowedTemperatureBasedCurrent.ContinuosChargeCurrent := MIN(AllowedTemperatureBasedCurrent.ContinuosChargeCurrent, tempCurrentLimits.ContinuosChargeCurrent);
	AllowedTemperatureBasedCurrent.ContinuosChargeCurrent := MIN(AllowedTemperatureBasedCurrent.PeakChargeCurrent, tempCurrentLimits.PeakChargeCurrent);
END_IF
END_METHOD

METHOD PRIVATE CalculateVoltageBasedCurrentLimits
VAR_INPUT
	minCellVoltage : REAL;
	maxCellVoltage : REAL;
	AllowedVoltageBasedCurrent : REFERENCE TO typSOF_CURRENT_LIMITS;
	CalculatedCurveValues : REFERENCE TO typSOF_CURVE;
	ConfigurationValues : REFERENCE TO typSOF_CONFIG;
END_VAR
IF (minCellVoltage <= ConfigurationValues.limitLowerCellVoltage_mV) THEN
	AllowedVoltageBasedCurrent.ContinuosDischargeCurrent := 0;
	AllowedVoltageBasedCurrent.PeakDischargeCurrent := 0;
ELSE
	IF (minCellVoltage <= ConfigurationValues.cutoffLowerCellVoltage_mV) THEN
		AllowedVoltageBasedCurrent.ContinuosDischargeCurrent := CalculatedCurveValues.slopeUpperCellVoltage * (minCellVoltage - ConfigurationValues.limitLowerCellVoltage_mV);
		AllowedVoltageBasedCurrent.PeakDischargeCurrent := AllowedVoltageBasedCurrent.ContinuosDischargeCurrent;
	ELSE
		AllowedVoltageBasedCurrent.ContinuosDischargeCurrent := ConfigurationValues.maximumDischargeCurrent_mA;
		AllowedVoltageBasedCurrent.PeakDischargeCurrent := ConfigurationValues.maximumDischargeCurrent_mA;
	END_IF
END_IF

IF (maxCellVoltage >= ConfigurationValues.limitUpperCellVoltage_mV) THEN
	AllowedVoltageBasedCurrent.ContinuosChargeCurrent := 0;
	AllowedVoltageBasedCurrent.PeakChargeCurrent := 0;
ELSE
	IF (maxCellVoltage <= ConfigurationValues.cutoffUpperCellVoltage_mV) THEN
		AllowedVoltageBasedCurrent.ContinuosChargeCurrent := CalculatedCurveValues.slopeLowerCellVoltage * (maxCellVoltage - ConfigurationValues.limitUpperCellVoltage_mV);
		AllowedVoltageBasedCurrent.PeakChargeCurrent := AllowedVoltageBasedCurrent.ContinuosChargeCurrent;
	ELSE
		AllowedVoltageBasedCurrent.ContinuosChargeCurrent := ConfigurationValues.maximumChargeCurrent_mA;
		AllowedVoltageBasedCurrent.PeakChargeCurrent := ConfigurationValues.maximumChargeCurrent_mA;
	END_IF
END_IF
END_METHOD

//FB_Init is always available implicitly and it is used primarily for initialization.
//The return value is not evaluated. For a specific influence, you can also declare the
//methods explicitly and provide additional code there with the standard initialization
//code. You can evaluate the return value.
METHOD FB_Init: BOOL
VAR_INPUT
    bInitRetains: BOOL; // TRUE: the retain variables are initialized (reset warm / reset cold)
    bInCopyCode: BOOL;  // TRUE: the instance will be copied to the copy code afterward (online change)   
END_VAR
CalculateCurves(CalculatedCurveValues := gvSOF.curveRecommandedOperatingCurrent,
				ConfigurationValues := gvSOF.SOF_Config);
END_METHOD

END_FUNCTION_BLOCK

// _750_8212_PFC200/Application/Utils/Pulse1Sec
FUNCTION_BLOCK Pulse1Sec
VAR_INPUT
	
END_VAR
VAR_OUTPUT
	Q : BOOL;
END_VAR
VAR
	init : BOOL;
	startTime : DWORD;
	deltaT : DWORD;
	QTrig : Standard.R_TRIG;
END_VAR

IF NOT init THEN
	startTime := T_PLC_MS();
	init := TRUE;
END_IF

Q := FALSE;
deltaT := T_PLC_MS() - startTime;

QTrig(CLK := deltaT >= 1000);

IF QTrig.Q THEN
	Q := TRUE;
	startTime := T_PLC_MS();
END_IF

END_FUNCTION_BLOCK

// _750_8212_PFC200/Application/BMS_String
FUNCTION_BLOCK BMS_String
VAR_INPUT
	//CellsData : REFERENCE TO typCELLS_VALUES;
	StringState : REFERENCE TO typSTRING_STATE;
END_VAR
VAR_OUTPUT
END_VAR
VAR
END_VAR

METHOD GetCurrentFlowDirection : eBMS_CURRENT_FLOW_STATE
VAR_INPUT
	StringCurrent : REAL;
END_VAR
IF STRING_CONFIG.BS_POSITIVE_DISCHARGE_CURRENT THEN
	IF (StringCurrent >= STRING_CONFIG.BS_REST_CURRENT_mA) THEN
		StringState.currentFlowState := eBMS_CURRENT_FLOW_STATE.DISCHARGING;
	ELSIF (StringCurrent <= -STRING_CONFIG.BS_REST_CURRENT_mA) THEN
		StringState.currentFlowState := eBMS_CURRENT_FLOW_STATE.CHARGING;
	ELSE
		StringState.currentFlowState := eBMS_CURRENT_FLOW_STATE.AT_REST;
	END_IF
ELSE
	IF (StringCurrent <= -STRING_CONFIG.BS_REST_CURRENT_mA) THEN
		StringState.currentFlowState := eBMS_CURRENT_FLOW_STATE.DISCHARGING;
	ELSIF (StringCurrent >= STRING_CONFIG.BS_REST_CURRENT_mA) THEN
		StringState.currentFlowState := eBMS_CURRENT_FLOW_STATE.CHARGING;
	ELSE
		StringState.currentFlowState := eBMS_CURRENT_FLOW_STATE.AT_REST;
	END_IF	
END_IF
END_METHOD

METHOD GetStringState : eBMS_CURRENT_FLOW_STATE
VAR_INPUT
END_VAR
GetStringState := StringState.currentFlowState;
END_METHOD

METHOD UpdateStringState
VAR_INPUT
	StringCurrent : REAL;
END_VAR

IF STRING_CONFIG.BS_POSITIVE_DISCHARGE_CURRENT THEN
	IF (StringCurrent >= STRING_CONFIG.BS_REST_CURRENT_mA) THEN
		StringState.currentFlowState := eBMS_CURRENT_FLOW_STATE.DISCHARGING;
		StringState.restTime := STRING_CONFIG.BS_RELAXATION_PERIOD;
	ELSIF (StringCurrent <= -STRING_CONFIG.BS_REST_CURRENT_mA) THEN
		StringState.currentFlowState := eBMS_CURRENT_FLOW_STATE.CHARGING;
		StringState.restTime := STRING_CONFIG.BS_RELAXATION_PERIOD;
	ELSE
		IF (StringState.restTime <= 0) THEN
			StringState.currentFlowState := eBMS_CURRENT_FLOW_STATE.AT_REST;
		ELSE
			StringState.currentFlowState := eBMS_CURRENT_FLOW_STATE.RELAXATION;
			StringState.restTime := StringState.restTime - 1000*TO_INT(gvBMS.Pulse1Sec.Q);
		END_IF
	END_IF
ELSE
	IF (StringCurrent <= -STRING_CONFIG.BS_REST_CURRENT_mA) THEN
		StringState.currentFlowState := eBMS_CURRENT_FLOW_STATE.DISCHARGING;
		StringState.restTime := STRING_CONFIG.BS_RELAXATION_PERIOD;
	ELSIF (StringCurrent >= STRING_CONFIG.BS_REST_CURRENT_mA) THEN
		StringState.currentFlowState := eBMS_CURRENT_FLOW_STATE.CHARGING;
		StringState.restTime := STRING_CONFIG.BS_RELAXATION_PERIOD;
	ELSE
		IF (StringState.restTime <= 0) THEN
			StringState.currentFlowState := eBMS_CURRENT_FLOW_STATE.AT_REST;
		ELSE
			StringState.currentFlowState := eBMS_CURRENT_FLOW_STATE.RELAXATION;
			StringState.restTime := StringState.restTime - 1000*TO_INT(gvBMS.Pulse1Sec.Q);
		END_IF
	END_IF	
END_IF
END_METHOD

END_FUNCTION_BLOCK

// _750_8212_PFC200/Application/Module
FUNCTION_BLOCK Module
VAR_INPUT
END_VAR
VAR_OUTPUT
END_VAR
VAR

END_VAR

END_FUNCTION_BLOCK

// _750_8212_PFC200/Application/BALANCING/BAL_Dukosi
FUNCTION_BLOCK BAL_Dukosi
VAR_INPUT
	DKS_BALCurrent : REFERENCE TO typCELL_BAL_CURRENT;
	DKS_BALControl : REFERENCE TO typCELL_CONTROL;
	DKS_BALStatus : REFERENCE TO typCELL_MEAS;
	DKS_CellVoltage : REFERENCE TO typCELL_VOLTAGE;
	DKS_MinMax : REFERENCE TO typMIN_MAX;
	balControl : REFERENCE TO typBALANCING_CONTROL;
END_VAR
VAR_OUTPUT
END_VAR
VAR
	//BalancingControl : BalancingControl(cellVoltage := gvCELLS.gvCellMeas.voltage, minMax := gvBMS.gvMinMax, balControl := gvBALANCING.gvBALANCING_CONTROL);
	idx : INT;
	EnableBalancingRTrig : Standard.R_TRIG;
	EnableBalancingFTrig : Standard.F_TRIG;
	enableBalancing : BOOL;
	balAlarmStop : BOOL;
	balNormalStop : BOOL;
	bal_State : typBAL_STATE;
	xInit : BOOL;
END_VAR

// 
// balAlarmStop := DKS_BALStatus.BalStatus.BAL_isStopError OR DKS_BALStatus.BalStatus.BAL_isStopOther OR DKS_BALStatus.BalStatus.BAL_isStopTemp;
// balNormalStop := DKS_BALStatus.BalStatus.BAL_IsStopCmd OR DKS_BALStatus.BalStatus.BAL_isStopTgtSoc OR DKS_BALStatus.BalStatus.BAL_IsStopTgtVolt OR DKS_BALStatus.BalStatus.BAL_isStopTgtWh;
// 
// EnableBalancingRTrig(CLK := EnBalancing);
// EnableBalancingFTrig(CLK := EnBalancing);
// 
// IF EnableBalancingRTrig.Q THEN
// 	enableBalancing := TRUE;
// END_IF
// 
// IF EnableBalancingFTrig.Q THEN
// 	enableBalancing := FALSE;
// END_IF
// 
// 
// IF EnableBalancing AND NOT DKS_BALStatus.BalStatus.BAL_isActive THEN
// 	BalancingControl.SetStateRequest(stateRequest := eBAL_STATE_REQUEST.BAL_STATE_GLOBAL_ENABLE_REQUEST);
// ELSE
// 	BalancingControl.SetStateRequest(stateRequest := eBAL_STATE_REQUEST.BAL_STATE_GLOBAL_DISABLE_REQUEST);
// END_IF
// 
// FOR idx := 1 TO STRING_CONFIG.BS_TOTAL_NR_OF_CELLS DO
// 	DKS_BALControl.BAL_Control[idx].ControlBits.BAL_enTgtVoltage := TO_BOOL(gvBALANCING.gvBALANCING_CONTROL.balancingState[idx]);
// END_FOR
// 
// 
// 
// gvBALANCING.gvBALANCING_CONTROL.enableBalancing := EnableBalancing AND NOT DKS_BALControl.BAL_Control
//

METHOD Activate : BOOL
VAR_INPUT

END_VAR
VAR
	cellBalancingCurrent : REAL;
	difference : INT;
	nrBalancedCells : INT;
	c : INT;
	finished : BOOL;
	minVoltage : REAL;
	balAlarm : BOOL;
	balTgtVoltageReached : BOOL;
END_VAR

finished := TRUE;
minVoltage := DKS_MinMax.minimumCellVoltage_mV;

FOR c := 1 TO STRING_CONFIG.BS_TOTAL_NR_OF_CELLS DO

	IF DKS_CellVoltage.cellVoltage_mV[c] > (minVoltage + bal_State.balancingThreshold) AND NOT (DKS_BALStatus.cellBalStatus[c].BalStatus.BAL_IsStopCmd OR 
	   DKS_BALStatus.cellBalStatus[c].BalStatus.BAL_isStopTgtSoc OR DKS_BALStatus.cellBalStatus[c].BalStatus.BAL_IsStopTgtVolt OR DKS_BALStatus.cellBalStatus[c].BalStatus.BAL_isStopTgtWh)  THEN
		balControl.balancingState[c] := 1;
		finished := FALSE;
		bal_State.balancingThreshold := balControl.threshold_mV;
		bal_state.active := TRUE;
		balControl.enableBalancing := TRUE;
		DKS_BALControl.BAL_Control[c].ControlBits.BAL_enTgtVoltage := TRUE;
		nrBalancedCells := nrBalancedCells + 1;
	ELSE
		balControl.balancingState[c] := 0;
	END_IF
END_FOR

balControl.nrBalancedCells := nrBalancedCells;

Activate := finished;
END_METHOD

METHOD BalancingAlarm : BOOL
VAR_INPUT
END_VAR
VAR
	idx : INT;
END_VAR
BalancingAlarm := FALSE;

FOR idx := 1 TO STRING_CONFIG.BS_TOTAL_NR_OF_CELLS DO
	IF DKS_BALStatus.cellBalStatus[idx].BalStatus.BAL_isStopError OR DKS_BALStatus.cellBalStatus[idx].BalStatus.BAL_isStopOther OR DKS_BALStatus.cellBalStatus[idx].BalStatus.BAL_isStopTemp THEN
		BalancingAlarm := TRUE;
		RETURN;
	END_IF
END_FOR
END_METHOD

METHOD CheckStateRequest : eBAL_RETURN
VAR_INPUT
	CurrentState : REFERENCE TO typBAL_STATE;
	stateRequest : eBAL_STATE_REQUEST;
END_VAR
IF (stateRequest = eBAL_STATE_REQUEST.BAL_STATE_ERROR_REQUEST) THEN
	CheckStateRequest := eBAL_RETURN.BAL_OK;
	RETURN;
END_IF

IF (stateRequest = eBAL_STATE_REQUEST.BAL_STATE_GLOBAL_ENABLE_REQUEST) THEN
	CurrentState.balancingGlobalAllowed := TRUE;
	CheckStateRequest := eBAL_RETURN.BAL_OK;
	RETURN;
END_IF

IF (stateRequest = eBAL_STATE_REQUEST.BAL_STATE_GLOBAL_DISABLE_REQUEST) THEN
	CurrentState.balancingGlobalAllowed := FALSE;
	CheckStateRequest := eBAL_RETURN.BAL_OK;
	RETURN;
END_IF

IF (stateRequest = eBAL_STATE_REQUEST.BAL_STATE_NO_BALANCING_REQUEST) OR (stateRequest = eBAL_STATE_REQUEST.BAL_STATE_ALLOWBALANCING_REQUEST) THEN
	CheckStateRequest := eBAL_RETURN.BAL_OK;
	RETURN;
END_IF

IF (CurrentState.stateRequest = eBAL_STATE_REQUEST.BAL_STATE_NO_REQUEST) THEN
	IF (stateRequest = eBAL_STATE_REQUEST.BAL_STATE_INIT_REQUEST) THEN
		IF (CurrentState.state = eBAL_STATE.BAL_STATEMACH_UNINITIALIZED) THEN
			CheckStateRequest := eBAL_RETURN.BAL_OK;
			RETURN;
		ELSE
			CheckStateRequest := eBAL_RETURN.BAL_ALREADY_INITIALIZED;
			RETURN;
		END_IF
	ELSE
		CheckStateRequest := eBAL_RETURN.BAL_ILLEGAL_REQUEST;
		RETURN;
	END_IF
ELSE
	CheckStateRequest := eBAL_RETURN.BAL_REQUEST_PENDING;
	RETURN;
END_IF
END_METHOD

METHOD Deactivate
VAR_INPUT
END_VAR
VAR
	c : INT;
END_VAR

FOR c := 1 TO STRING_CONFIG.BS_TOTAL_NR_OF_CELLS DO
	balControl.balancingState[c] := 0;
	DKS_BALControl.BAL_Control[c].ControlBits.BAL_enTgtVoltage := FALSE;
END_FOR
balControl.nrBalancedCells := 0;
balControl.enableBalancing := 0;
bal_State.active := FALSE;
END_METHOD

METHOD ProcessState_Balancing
VAR_INPUT
	stateRequest : eBAL_STATE_REQUEST;
END_VAR
IF (stateRequest = eBAL_STATE_REQUEST.BAL_STATE_NO_BALANCING_REQUEST) THEN
	bal_State.balancingAllowed := FALSE;
END_IF

IF (stateRequest = eBAL_STATE_REQUEST.BAL_STATE_ALLOWBALANCING_REQUEST) THEN
	bal_State.balancingAllowed := TRUE;
END_IF

IF (BalancingAlarm() = TRUE) THEN
	bal_State.balancingAllowed := FALSE;
END_IF

IF (bal_State.balancingGlobalAllowed = FALSE) THEN
	IF (bal_State.active) THEN
		Deactivate();
	END_IF
	bal_State.active := FALSE;
	bal_State.state := eBAL_STATE.BAL_STATEMACH_BALANCE;
	bal_State.substate := eBAL_SUB_STATE.BAL_ENTRY;
	RETURN;
END_IF

IF (bal_State.substate = eBAL_SUB_STATE.BAL_ENTRY) THEN
	IF (bal_State.balancingGlobalAllowed = FALSE) THEN
		IF (bal_State.active) THEN
			Deactivate();
		END_IF
		bal_State.active := FALSE;
		bal_State.state := eBAL_STATE.BAL_STATEMACH_BALANCE;
		bal_State.substate := eBAL_SUB_STATE.BAL_ENTRY;
	ELSE
		bal_State.substate := eBAL_SUB_STATE.BAL_CHECK_LOWEST_VOLTAGE;
	END_IF
ELSIF (bal_State.substate = eBAL_SUB_STATE.BAL_CHECK_LOWEST_VOLTAGE) THEN
	bal_State.substate := eBAL_SUB_STATE.BAL_CHECK_CURRENT;
	IF (DKS_MinMax.minimumCellVoltage_mV <= BALANCING_CONFIG.BAL_LOWER_VOLTAGE_LIMIT_mV) OR 
	    (DKS_MinMax.maximumTemperature_degC >= BALANCING_CONFIG.BAL_UPPER_TEMPERATURE_LIMIT_degC) THEN
		IF (bal_State.active) THEN
			Deactivate();
		END_IF
		bal_State.active := FALSE;
		bal_State.state := eBAL_STATE.BAL_STATEMACH_CHECK_BALANCING;
		bal_State.substate := eBAL_SUB_STATE.BAL_ENTRY;
	END_IF
	RETURN;
ELSIF (bal_State.substate = eBAL_SUB_STATE.BAL_CHECK_CURRENT) THEN
	IF (gvBMS.Fb_String.GetStringState() = eBMS_CURRENT_FLOW_STATE.AT_REST) THEN
		bal_State.substate := eBAL_SUB_STATE.BAL_ACTIVATE_BALANCING;
	ELSE
		IF (bal_State.active) THEN
			Deactivate();
		END_IF
		bal_State.active := FALSE;
		bal_State.state := eBAL_STATE.BAL_STATEMACH_CHECK_BALANCING;
		bal_State.substate := eBAL_SUB_STATE.BAL_ENTRY;	
	END_IF
	RETURN;
ELSIF (bal_State.substate = eBAL_SUB_STATE.BAL_ACTIVATE_BALANCING) THEN
	IF (bal_State.balancingGlobalAllowed = FALSE) THEN
		IF (bal_State.active) THEN
			Deactivate();
		END_IF
		bal_State.active := FALSE;
		bal_State.state := eBAL_STATE.BAL_STATEMACH_BALANCE;
		bal_State.substate := eBAL_SUB_STATE.BAL_ENTRY;
	ELSE
		IF (Activate() = TRUE) THEN
			bal_State.balancingThreshold := balControl.threshold_mV + BALANCING_CONFIG.BAL_HYSTERESIS_mV;
			bal_State.state := eBAL_STATE.BAL_STATEMACH_CHECK_BALANCING;
			bal_State.substate := eBAL_SUB_STATE.BAL_ENTRY;
		ELSE
			bal_State.state := eBAL_STATE.BAL_STATEMACH_BALANCE;
			bal_State.substate := eBAL_SUB_STATE.BAL_ENTRY;
		END_IF
	END_IF
	RETURN;
END_IF
END_METHOD

METHOD ProcessState_CheckBalancing
VAR_INPUT
	stateRequest : eBAL_STATE_REQUEST;
END_VAR
IF (stateRequest = eBAL_STATE_REQUEST.BAL_STATE_NO_BALANCING_REQUEST) THEN
	bal_State.balancingAllowed := FALSE;
END_IF

IF (stateRequest = eBAL_STATE_REQUEST.BAL_STATE_ALLOWBALANCING_REQUEST) THEN
	bal_State.balancingAllowed := TRUE;
END_IF

IF ((bal_State.balancingAllowed = FALSE) OR (bal_State.balancingGlobalAllowed = FALSE)) THEN
	Deactivate();
	bal_State.active := FALSE;
ELSE
	IF (gvBMS.Fb_String.GetStringState() = eBMS_CURRENT_FLOW_STATE.AT_REST) THEN
		bal_State.state := eBAL_STATE.BAL_STATEMACH_BALANCE;
		bal_State.substate := eBAL_SUB_STATE.BAL_ENTRY;
	END_IF
END_IF
END_METHOD

METHOD Run
VAR_INPUT
END_VAR
VAR
	stateRequest : eBAL_STATE_REQUEST;
	
END_VAR
IF NOT xInit THEN
	bal_State.state := eBAL_STATE.BAL_STATEMACH_CHECK_BALANCING;
	xInit := true;
END_IF

//stateRequest := eBAL_STATE_REQUEST.BAL_STATE_NO_REQUEST;

CASE bal_State.state OF
	
	eBAL_STATE.BAL_STATEMACH_CHECK_BALANCING:
		stateRequest := TransferStateRequest(bal_State);
		ProcessState_CheckBalancing(stateRequest);
		
	eBAL_STATE.BAL_STATEMACH_BALANCE:
		stateRequest := TransferStateRequest(bal_State);
		ProcessState_Balancing(stateRequest);
		
END_CASE
END_METHOD

METHOD SetStateRequest : eBAL_RETURN
VAR_INPUT
	stateRequest : eBAL_STATE_REQUEST;
END_VAR
VAR
	retVal : eBAL_RETURN;
END_VAR
SetStateRequest := eBAL_RETURN.BAL_OK;

retVal := CheckStateRequest(bal_State, stateRequest);

IF retVal = eBAL_RETURN.BAL_OK THEN
	bal_State.stateRequest := stateRequest;
END_IF

SetStateRequest := retVal;
END_METHOD

METHOD TransferStateRequest : eBAL_STATE_REQUEST
VAR_INPUT
	currentState : REFERENCE TO typBAL_STATE;
END_VAR
VAR
	retVal : eBAL_STATE_REQUEST;

END_VAR
retVal := eBAL_STATE_REQUEST.BAL_STATE_NO_REQUEST;

retVal := currentState.stateRequest;
currentState.stateRequest := eBAL_STATE_REQUEST.BAL_STATE_NO_REQUEST;

TransferStateRequest := retVal;
END_METHOD

END_FUNCTION_BLOCK

// _750_8212_PFC200/Application/BMS/StringMinMax
FUNCTION_BLOCK StringMinMax
VAR_INPUT
	MinMaxTable : REFERENCE TO typMIN_MAX;
	//CellsData : REFERENCE TO typCELLS_VALUES;
END_VAR
VAR_OUTPUT
END_VAR
VAR
END_VAR

METHOD PRIVATE CalculateDyeTemperatureMinMaxAverage : eRET_VAL
VAR_INPUT
	CellDyeTemperature : REFERENCE TO typCELL_DYE_TEMPERATURE;
END_VAR
VAR
	_ret_val : eRET_VAL;
	_nrValidCellsDyeTemperature : INT;
	_min : REAL;
	_max : REAL;
	_sum : REAL;
	c : INT;
	m : INT;
END_VAR
_ret_val := eRET_VAL.STD_OK;
_nrValidCellsDyeTemperature := 0;


	FOR c := 1 TO STRING_CONFIG.BS_TOTAL_NR_OF_CELLS DO
		m := TO_INT(c/STRING_CONFIG.BS_MAX_NR_OF_CELLS_PER_MODULE) + 1;
		IF (SHR(CellDyeTemperature.invalidCellDyeTemperature[m], c) AND 16#1) = 0 THEN
			_nrValidCellsDyeTemperature := _nrValidCellsDyeTemperature + 1;
			_sum := _sum + CellDyeTemperature.cellDyeTemperature_deg[c];
			
			IF CellDyeTemperature.cellDyeTemperature_deg[c] < _min THEN
				_min := CellDyeTemperature.cellDyeTemperature_deg[c];
			END_IF
			
			IF CellDyeTemperature.cellDyeTemperature_deg[c] > _max THEN
				_max := CellDyeTemperature.cellDyeTemperature_deg[c];
			END_IF	
		END_IF
	END_FOR


MinMaxTable.minimumDyeTemperature_degC := _min;
MinMaxTable.maximumDyeTemperature_degC := _max;
MinMaxTable.validMeasuredCellDyeTemperatures := _nrValidCellsDyeTemperature;


IF _nrValidCellsDyeTemperature > 0 THEN
	MinMaxTable.averageDyeTemperature_degC := _sum/_nrValidCellsDyeTemperature;
ELSE
	MinMaxTable.averageDyeTemperature_degC := 0;
	_ret_val := eRET_VAL.STD_NOT_OK;	
END_IF

CalculateDyeTemperatureMinMaxAverage := _ret_val;
END_METHOD

METHOD PRIVATE CalculateTemperatureMinMaxAverage : eRET_VAL
VAR_INPUT
	CellTemperature : REFERENCE TO typCELL_TEMPERATURE;
END_VAR
VAR

	_ret_val : eRET_VAL;
	_nrValidCellsTemperature : INT;
	_min : REAL;
	_max : REAL;
	_sum : REAL;
	c : INT;
	m : INT;
END_VAR
_ret_val := eRET_VAL.STD_OK;
_nrValidCellsTemperature := 0;

FOR c := 1 TO STRING_CONFIG.BS_TOTAL_NR_OF_CELLS DO
	m := TO_INT(c/STRING_CONFIG.BS_MAX_NR_OF_CELLS_PER_MODULE) + 1;
	IF (SHR(CellTemperature.invalidCellTemperature[m], c) AND 16#1) = 0 THEN
		_nrValidCellsTemperature := _nrValidCellsTemperature + 1;
		_sum := _sum + CellTemperature.cellTemperature_deg[c];
		
		IF CellTemperature.cellTemperature_deg[c] < _min THEN
			_min := CellTemperature.cellTemperature_deg[c];
		END_IF
		
		IF CellTemperature.cellTemperature_deg[c] > _max THEN
			_max := CellTemperature.cellTemperature_deg[c];
		END_IF
		
	END_IF
END_FOR


MinMaxTable.minimumTemperature_degC := _min;
MinMaxTable.maximumTemperature_degC := _max;
MinMaxTable.validMeasuredCellTemperatures := _nrValidCellsTemperature;


IF _nrValidCellsTemperature > 0 THEN
	MinMaxTable.averageTemperature_degC := _sum/_nrValidCellsTemperature;
ELSE
	MinMaxTable.averageTemperature_degC := 0;
	_ret_val := eRET_VAL.STD_NOT_OK;	
END_IF



CalculateTemperatureMinMaxAverage := _ret_val;
END_METHOD

METHOD PRIVATE CalculateVoltageMinMaxAverage : eRET_VAL
VAR_INPUT
	CellVoltage : REFERENCE TO typCELL_VOLTAGE;
END_VAR
VAR
	c : INT;
	m : INT;
	_ret_val : eRET_VAL;
	_nrValidCellsVoltage : INT;
	_min : REAL;
	_max : REAL;
	_sum : DINT;

END_VAR
_ret_val := eRET_VAL.STD_OK;
_nrValidCellsVoltage := 0;

FOR c := 1 TO STRING_CONFIG.BS_TOTAL_NR_OF_CELLS DO
	m := TO_INT(c/STRING_CONFIG.BS_MAX_NR_OF_CELLS_PER_MODULE) + 1;
	IF (SHR(CellVoltage.invalidCellVoltage[m], c) AND 16#1) = 0 THEN
		_nrValidCellsVoltage := _nrValidCellsVoltage + 1;
		_sum := _sum + CellVoltage.cellVoltage_mV[c];
		
		IF CellVoltage.cellVoltage_mV[c] < _min THEN
			_min := CellVoltage.cellVoltage_mV[c];
		END_IF
		
		IF CellVoltage.cellVoltage_mV[c] > _max THEN
			_max := CellVoltage.cellVoltage_mV[c];
		END_IF
		
	END_IF
END_FOR

MinMaxTable.minimumCellVoltage_mV := _min;
MinMaxTable.maximumCellVoltage_mV := _max;
MinMaxTable.validMeasuredCellVoltages := _nrValidCellsVoltage;

IF _nrValidCellsVoltage > 0 THEN
	MinMaxTable.averageCellVoltage_mV := TO_REAL(_sum/_nrValidCellsVoltage);
ELSE
	MinMaxTable.averageCellVoltage_mV := 0;
	_ret_val := eRET_VAL.STD_NOT_OK;	
END_IF

CellVoltage.stringVoltage_mV := _sum;

CalculateVoltageMinMaxAverage := _ret_val;
END_METHOD

METHOD PRIVATE CheckDyeTemperatureSpread : eRET_VAL
VAR_INPUT
	CellDyeTemperature : REFERENCE TO typCELL_DYE_TEMPERATURE;
END_VAR
VAR
	c : INT;
	m : INT;
	_ret_val : eRET_VAL;
END_VAR
VAR CONSTANT
	dat : ULINT := 1;
END_VAR
_ret_val := eRET_VAL.STD_OK;
CellDyeTemperature.nrValidCellDyeTemperatures := 0;

FOR m := 1 TO STRING_CONFIG.BS_NR_OF_MODULES DO
	CellDyeTemperature.invalidCellDyeTemperature[m] := 0;
END_FOR

FOR c := 1 TO STRING_CONFIG.BS_TOTAL_NR_OF_CELLS DO
	m := TO_INT(c/STRING_CONFIG.BS_MAX_NR_OF_CELLS_PER_MODULE) + 1;
	IF (SHR(CellDyeTemperature.invalidCellDyeTemperature[m], c) AND 16#1) = 0 THEN
		IF ABS(CellDyeTemperature.cellDyeTemperature_deg[c] - MinMaxTable.averageDyeTemperature_degC) > BAT_CELL_CONFIG.CELL_DYE_TEMPERATURE_SPREAD_TOLERANCE THEN
			_ret_val := eRET_VAL.STD_NOT_OK;
			CellDyeTemperature.invalidCellDyeTemperature[m] := CellDyeTemperature.invalidCellDyeTemperature[m] OR SHR(dat, c);
		ELSE
			CellDyeTemperature.nrValidCellDyeTemperatures := CellDyeTemperature.nrValidCellDyeTemperatures + 1;
		END_IF	
	END_IF
END_FOR


CheckDyeTemperatureSpread := _ret_val;
END_METHOD

METHOD PRIVATE CheckTemperatureSpread : eRET_VAL
VAR_INPUT
	CellTemperature : REFERENCE TO typCELL_TEMPERATURE;
END_VAR
VAR
	m : INT;
	c : INT;
	_ret_val : eRET_VAL;
END_VAR
VAR CONSTANT
	dat : ULINT := 1;
END_VAR
_ret_val := eRET_VAL.STD_OK;
CellTemperature.nrValidCellTemperatures := 0;

FOR m := 1 TO STRING_CONFIG.BS_NR_OF_MODULES DO
	CellTemperature.invalidCellTemperature[m] := 0;
END_FOR

FOR c := 1 TO STRING_CONFIG.BS_TOTAL_NR_OF_CELLS DO
	m := TO_INT(c/STRING_CONFIG.BS_MAX_NR_OF_CELLS_PER_MODULE) + 1;
	IF (SHR(CellTemperature.invalidCellTemperature[m], c) AND 16#1) = 0 THEN
		IF ABS(CellTemperature.cellTemperature_deg[c] - MinMaxTable.averageTemperature_degC) > BAT_CELL_CONFIG.CELL_TEMPERATURE_SPREAD_TOLERANCE THEN
			_ret_val := eRET_VAL.STD_NOT_OK;
			CellTemperature.invalidCellTemperature[m] := CellTemperature.invalidCellTemperature[m] OR SHR(dat, c);
		ELSE
			CellTemperature.nrValidCellTemperatures := CellTemperature.nrValidCellTemperatures + 1;
		END_IF	
	END_IF
END_FOR


CheckTemperatureSpread := _ret_val;
END_METHOD

METHOD PRIVATE CheckVoltageSpread : eRET_VAL
VAR_INPUT
	CellVoltage : REFERENCE TO typCELL_VOLTAGE;
END_VAR
VAR
	c : INT;
	m : INT;
	_ret_val : eRET_VAL;
END_VAR
VAR CONSTANT
	dat : ULINT := 1;
END_VAR
_ret_val := eRET_VAL.STD_OK;
CellVoltage.nrValidCellVoltages := 0;

FOR m := 1 TO STRING_CONFIG.BS_NR_OF_MODULES DO
	CellVoltage.invalidCellVoltage[m] := 0;
END_FOR

FOR c := 1 TO STRING_CONFIG.BS_TOTAL_NR_OF_CELLS DO
	m := TO_INT(c/STRING_CONFIG.BS_MAX_NR_OF_CELLS_PER_MODULE) + 1;
	IF (SHR(CellVoltage.invalidCellVoltage[m], c) AND 16#1) = 0 THEN
		IF ABS(CellVoltage.cellVoltage_mV[c] - MinMaxTable.averageCellVoltage_mV) > BAT_CELL_CONFIG.CELL_VOLTAGE_SPREAD_TOLERANCE THEN
			_ret_val := eRET_VAL.STD_NOT_OK;
			CellVoltage.invalidCellVoltage[m] := CellVoltage.invalidCellVoltage[m] OR SHR(dat, c);
		ELSE
			CellVoltage.nrValidCellVoltages := CellVoltage.nrValidCellVoltages + 1;
		END_IF	
	END_IF
END_FOR	


CheckVoltageSpread := _ret_val;
END_METHOD

METHOD Main
VAR_INPUT
END_VAR
ValidateCellTemperature(gvCELLS.gvCellTemp.temperature);
ValidateCellVoltage(gvCELLS.gvCellMeas.voltage);
ValidateCellDyeTemperature(gvCELLS.gvCellTemp.dyeTemperature);
END_METHOD

METHOD ValidateCellDyeTemperature
VAR_INPUT
	CellDyeTemperature : REFERENCE TO typCELL_DYE_TEMPERATURE;
END_VAR
CalculateDyeTemperatureMinMaxAverage(CellDyeTemperature);

IF (eRET_VAL.STD_NOT_OK = CheckDyeTemperatureSpread(CellDyeTemperature)) THEN
	CalculateDyeTemperatureMinMaxAverage(CellDyeTemperature);
END_IF
END_METHOD

METHOD ValidateCellTemperature
VAR_INPUT
	CellTemperature : REFERENCE TO typCELL_TEMPERATURE;
END_VAR
CalculateTemperatureMinMaxAverage(CellTemperature);

IF (eRET_VAL.STD_NOT_OK = CheckTemperatureSpread(CellTemperature)) THEN
	CalculateTemperatureMinMaxAverage(CellTemperature);
END_IF
END_METHOD

METHOD ValidateCellVoltage
VAR_INPUT
	CellVoltage : REFERENCE TO typCELL_VOLTAGE;
END_VAR
CalculateVoltageMinMaxAverage(CellVoltage);

IF (eRET_VAL.STD_NOT_OK = CheckVoltageSpread(CellVoltage)) THEN
	CalculateVoltageMinMaxAverage(CellVoltage);
END_IF
END_METHOD

END_FUNCTION_BLOCK

// _750_8212_PFC200/Application/BMSUtils/GetSOCFromVoltage
FUNCTION GetSOCFromVoltage : REAL
VAR_INPUT
	voltage_mV : REAL;
END_VAR
VAR
	_socPercent : REAL;
	_betweenHigh : UINT;
	_betweenLow : UINT;
	idx : UINT;
END_VAR

_socPercent := 0.5;
_betweenHigh := 0;
_betweenLow := 0;

FOR idx := 1 TO BAT_CELL_CONFIG.stateOfChargeLookupTableSize DO
	IF voltage_mV < BAT_CELL_CONFIG.stateOfChargeLookupTable[idx].Voltage THEN
		_betweenHigh := idx;
		_betweenLow := idx + 1;
	END_IF;	
END_FOR

IF (NOT ((_betweenHigh = 0 AND _betweenLow = 0) OR (_betweenLow >= BAT_CELL_CONFIG.stateOfChargeLookupTableSize))) THEN
	_socPercent := MATH_LinearInterpolation(X1 := TO_REAL(BAT_CELL_CONFIG.stateOfChargeLookupTable[_betweenLow].Voltage),
											Y1 := BAT_CELL_CONFIG.stateOfChargeLookupTable[_betweenLow].SOC,
											X2 := TO_REAL(BAT_CELL_CONFIG.stateOfChargeLookupTable[_betweenHigh].Voltage),
											Y2 := BAT_CELL_CONFIG.stateOfChargeLookupTable[_betweenHigh].SOC,
											X  := voltage_mV);
ELSIF (_betweenLow >= BAT_CELL_CONFIG.stateOfChargeLookupTableSize) THEN
	_socPercent := 0;
ELSE
	_socPercent := 100;																					
END_IF

END_FUNCTION

